# B&R Automation Studio project NAEUL004C00R13L518F00 (part 15)

#### Act_OptP0910WriteDO.st
```iecst
ACTION Act_OptP0910WriteDO:

	//TL Safety Relay
	IF tyP0910GenOut.tyGenOut.tyBtnSafetyRst.bRtCompl = TRUE THEN
		IF tyP0910GenOut.tyGenOut.tyBtnSafetyRst.bValue = TRUE THEN
			eRstErrAct	:= RstErrActSetSafetyRlyRst;

			IF p_eRstErrStat = RstErrActSetSafetyRlyRst AND p_eRstErrStatus = Done THEN
				eRstErrAct	:= RstErrActIdle;

				tyP0910GenOut.tyGenOut.tyBtnSafetyRst.bRtCompl	:= FALSE;
			END_IF
		ELSE
			eRstErrAct	:= RstErrActRstSafetyRlyRst;

			IF p_eRstErrStat = RstErrActRstSafetyRlyRst AND p_eRstErrStatus = Done THEN
				eRstErrAct	:= RstErrActIdle;

				tyP0910GenOut.tyGenOut.tyBtnSafetyRst.bRtCompl	:= FALSE;
			END_IF

		END_IF
	END_IF

	// TL Green
	IF tyP0910GenOut.tyGenOut.tyBtnTLGreen.bRtCompl = TRUE THEN
		IF tyP0910GenOut.tyGenOut.tyBtnTLGreen.bValue = TRUE THEN
			eTLBuzAct	:= TLBuzActSetGreen;

			IF p_eTLBuzStat = TLBuzActSetGreen AND p_eTLBuzStatus = Done THEN
				eTLBuzAct	:= TLBuzActIdle;

				tyP0910GenOut.tyGenOut.tyBtnTLGreen.bRtCompl	:= FALSE;
			END_IF
		ELSE
			eTLBuzAct	:= TLBuzActRstGreen;

			IF p_eTLBuzStat = TLBuzActRstGreen AND p_eTLBuzStatus = Done THEN
				eTLBuzAct	:= TLBuzActIdle;

				tyP0910GenOut.tyGenOut.tyBtnTLGreen.bRtCompl	:= FALSE;
			END_IF

		END_IF
	END_IF

	//TL Amber
	IF tyP0910GenOut.tyGenOut.tyBtnTLAmber.bRtCompl = TRUE THEN
		IF tyP0910GenOut.tyGenOut.tyBtnTLAmber.bValue = TRUE THEN
			IF p_tyNtParamCurr.eCustomerReq = Siemens THEN
				eTLBuzAct	:= TLBuzActSetWhite;
				IF p_eTLBuzStat = TLBuzActSetWhite AND p_eTLBuzStatus = Done THEN
					eTLBuzAct	:= TLBuzActIdle;
				END_IF
			ELSE
				eTLBuzAct	:= TLBuzActSetAmber;
				IF p_eTLBuzStat = TLBuzActSetAmber AND p_eTLBuzStatus = Done THEN
					eTLBuzAct	:= TLBuzActIdle;

					tyP0910GenOut.tyGenOut.tyBtnTLAmber.bRtCompl	:= FALSE;
				END_IF
			END_IF
		ELSE
			IF p_tyNtParamCurr.eCustomerReq = Siemens THEN
				eTLBuzAct	:= TLBuzActRstWhite;
				IF p_eTLBuzStat = TLBuzActRstWhite AND p_eTLBuzStatus = Done THEN
					eTLBuzAct	:= TLBuzActIdle;

					tyP0910GenOut.tyGenOut.tyBtnTLAmber.bRtCompl	:= FALSE;
				END_IF
			ELSE
				eTLBuzAct	:= TLBuzActRstAmber;
				IF p_eTLBuzStat = TLBuzActRstAmber AND p_eTLBuzStatus = Done THEN
					eTLBuzAct	:= TLBuzActIdle;

					tyP0910GenOut.tyGenOut.tyBtnTLAmber.bRtCompl	:= FALSE;
				END_IF
			END_IF
		END_IF
	END_IF

	//TL Red
	IF tyP0910GenOut.tyGenOut.tyBtnTLRed.bRtCompl = TRUE THEN
		IF tyP0910GenOut.tyGenOut.tyBtnTLRed.bValue = TRUE THEN
			eTLBuzAct	:= TLBuzActSetRed;

			IF p_eTLBuzStat = TLBuzActSetRed AND p_eTLBuzStatus = Done THEN
				eTLBuzAct	:= TLBuzActIdle;

				tyP0910GenOut.tyGenOut.tyBtnTLRed.bRtCompl	:= FALSE;
			END_IF
		ELSE
			eTLBuzAct	:= TLBuzActRstRed;

			IF p_eTLBuzStat = TLBuzActRstRed AND p_eTLBuzStatus = Done THEN
				eTLBuzAct	:= TLBuzActIdle;

				tyP0910GenOut.tyGenOut.tyBtnTLRed.bRtCompl	:= FALSE;
			END_IF

		END_IF
	END_IF

	//TL Buzzer
	IF tyP0910GenOut.tyGenOut.tyBtnBuzzer.bRtCompl = TRUE THEN
		IF tyP0910GenOut.tyGenOut.tyBtnBuzzer.bValue = TRUE THEN
			eTLBuzAct	:= TLBuzActSetBuz;

			IF p_eTLBuzStat = TLBuzActSetBuz AND p_eTLBuzStatus = Done THEN
				eTLBuzAct	:= TLBuzActIdle;

				tyP0910GenOut.tyGenOut.tyBtnBuzzer.bRtCompl	:= FALSE;
			END_IF
		ELSE
			eTLBuzAct	:= TLBuzActRstBuz;

			IF p_eTLBuzStat = TLBuzActRstBuz AND p_eTLBuzStatus = Done THEN
				eTLBuzAct	:= TLBuzActIdle;

				tyP0910GenOut.tyGenOut.tyBtnBuzzer.bRtCompl	:= FALSE;
			END_IF

		END_IF
	END_IF

	//Oven Info A
	IF tyP0910GenOut.tyOven.tyBtnOvenInfoA.bRtCompl = TRUE THEN
		IF tyP0910GenOut.tyOven.tyBtnOvenInfoA.bValue = TRUE THEN
			eOvenInfoAAct	:= OvenInfoActSetOvenAllow;

			IF p_eOvenInfoAStat = OvenInfoActSetOvenAllow AND p_eOvenInfoAStatus = Done THEN
				eOvenInfoAAct	:= OvenInfoActIdle;

				tyP0910GenOut.tyOven.tyBtnOvenInfoA.bRtCompl	:= FALSE;
			END_IF
		ELSE
			eOvenInfoAAct	:= OvenInfoActRstOvenAllow;

			IF p_eOvenInfoAStat = OvenInfoActRstOvenAllow AND p_eOvenInfoAStatus = Done THEN
				eOvenInfoAAct	:= OvenInfoActIdle;

				tyP0910GenOut.tyOven.tyBtnOvenInfoA.bRtCompl	:= FALSE;
			END_IF

		END_IF
	END_IF

	//Oven Info B
	IF tyP0910GenOut.tyOven.tyBtnOvenInfoB.bRtCompl = TRUE THEN
		IF tyP0910GenOut.tyOven.tyBtnOvenInfoB.bValue = TRUE THEN
			eOvenInfoBAct	:= OvenInfoActSetOvenAllow;

			IF p_eOvenInfoBStat = OvenInfoActSetOvenAllow AND p_eOvenInfoBStatus = Done THEN
				eOvenInfoBAct	:= OvenInfoActIdle;

				tyP0910GenOut.tyOven.tyBtnOvenInfoB.bRtCompl	:= FALSE;
			END_IF
		ELSE
			eOvenInfoBAct	:= OvenInfoActRstOvenAllow;

			IF p_eOvenInfoBStat = OvenInfoActRstOvenAllow AND p_eOvenInfoBStatus = Done THEN
				eOvenInfoBAct	:= OvenInfoActIdle;

				tyP0910GenOut.tyOven.tyBtnOvenInfoB.bRtCompl	:= FALSE;
			END_IF

		END_IF
	END_IF

	//Bypass Open Limit Sen
	IF tyP0910GenOut.tyMagAW.tyBtnMagAWOpenLimByp1.bRtCompl = TRUE THEN

		IF tyP0910GenOut.tyMagAW.tyBtnMagAWOpenLimByp1.bValue = TRUE THEN
			bMagAWOpenLimByp1 := TRUE;
			tyP0910GenOut.tyMagAW.tyBtnMagAWOpenLimByp1.bRtCompl := FALSE;
		ELSE
			bMagAWOpenLimByp1 := FALSE;
			tyP0910GenOut.tyMagAW.tyBtnMagAWOpenLimByp1.bRtCompl := FALSE;
		END_IF
	END_IF

	IF tyP0910GenOut.tyMagAW.tyBtnMagAWOpenLimByp2.bRtCompl = TRUE THEN

		IF tyP0910GenOut.tyMagAW.tyBtnMagAWOpenLimByp2.bValue = TRUE THEN
			bMagAWOpenLimByp2 := TRUE;
			tyP0910GenOut.tyMagAW.tyBtnMagAWOpenLimByp2.bRtCompl := FALSE;
		ELSE
			bMagAWOpenLimByp2 := FALSE;
			tyP0910GenOut.tyMagAW.tyBtnMagAWOpenLimByp2.bRtCompl := FALSE;
		END_IF
	END_IF

	IF tyP0910GenOut.tyMagAW.tyBtnMagAWOpenLimByp3.bRtCompl = TRUE THEN

		IF tyP0910GenOut.tyMagAW.tyBtnMagAWOpenLimByp3.bValue = TRUE THEN
			bMagAWOpenLimByp3 := TRUE;
			tyP0910GenOut.tyMagAW.tyBtnMagAWOpenLimByp3.bRtCompl := FALSE;
		ELSE
			bMagAWOpenLimByp3 := FALSE;
			tyP0910GenOut.tyMagAW.tyBtnMagAWOpenLimByp3.bRtCompl := FALSE;
		END_IF
	END_IF

	IF tyP0910GenOut.tyMagAW.tyBtnMagAWOpenLimByp4.bRtCompl = TRUE THEN

		IF tyP0910GenOut.tyMagAW.tyBtnMagAWOpenLimByp4.bValue = TRUE THEN
			bMagAWOpenLimByp4 := TRUE;
			tyP0910GenOut.tyMagAW.tyBtnMagAWOpenLimByp4.bRtCompl := FALSE;
		ELSE
			bMagAWOpenLimByp4 := FALSE;
			tyP0910GenOut.tyMagAW.tyBtnMagAWOpenLimByp4.bRtCompl := FALSE;
		END_IF
	END_IF

	//Select Small Mag Open Limit Sen
	IF tyP0910GenOut.tyMagAW.tyBtnSmallMagAWLimSen1.bRtCompl = TRUE THEN

		IF tyP0910GenOut.tyMagAW.tyBtnSmallMagAWLimSen1.bValue = TRUE THEN
			bSmallMagLimSen1 := TRUE;
			tyP0910GenOut.tyMagAW.tyBtnSmallMagAWLimSen1.bRtCompl := FALSE;
		ELSE
			bSmallMagLimSen1 := FALSE;
			tyP0910GenOut.tyMagAW.tyBtnSmallMagAWLimSen1.bRtCompl := FALSE;
		END_IF
	END_IF

	IF tyP0910GenOut.tyMagAW.tyBtnSmallMagAWLimSen2.bRtCompl = TRUE THEN

		IF tyP0910GenOut.tyMagAW.tyBtnSmallMagAWLimSen2.bValue = TRUE THEN
			bSmallMagLimSen2 := TRUE;
			tyP0910GenOut.tyMagAW.tyBtnSmallMagAWLimSen2.bRtCompl := FALSE;
		ELSE
			bSmallMagLimSen2 := FALSE;
			tyP0910GenOut.tyMagAW.tyBtnSmallMagAWLimSen2.bRtCompl := FALSE;
		END_IF
	END_IF

	IF tyP0910GenOut.tyMagAW.tyBtnSmallMagAWLimSen3.bRtCompl = TRUE THEN

		IF tyP0910GenOut.tyMagAW.tyBtnSmallMagAWLimSen3.bValue = TRUE THEN
			bSmallMagLimSen3 := TRUE;
			tyP0910GenOut.tyMagAW.tyBtnSmallMagAWLimSen3.bRtCompl := FALSE;
		ELSE
			bSmallMagLimSen3 := FALSE;
			tyP0910GenOut.tyMagAW.tyBtnSmallMagAWLimSen3.bRtCompl := FALSE;
		END_IF
	END_IF

	IF tyP0910GenOut.tyMagAW.tyBtnSmallMagAWLimSen4.bRtCompl = TRUE THEN

		IF tyP0910GenOut.tyMagAW.tyBtnSmallMagAWLimSen4.bValue = TRUE THEN
			bSmallMagLimSen4 := TRUE;
			tyP0910GenOut.tyMagAW.tyBtnSmallMagAWLimSen4.bRtCompl := FALSE;
		ELSE
			bSmallMagLimSen4 := FALSE;
			tyP0910GenOut.tyMagAW.tyBtnSmallMagAWLimSen4.bRtCompl := FALSE;
		END_IF
	END_IF

//	IF tyP0910GenOut.tyGenOutCurtainSen.tyBtnRstCurtainSen.bRtCompl = TRUE THEN
//
//		IF tyP0910GenOut.tyGenOutCurtainSen.tyBtnRstCurtainSen.bValue = TRUE THEN
//			bSafetyCurtainReset := TRUE;
//			tyP0910GenOut.tyGenOutCurtainSen.tyBtnRstCurtainSen.bRtCompl := FALSE;
//		ELSE
//			bSafetyCurtainReset := FALSE;
//			tyP0910GenOut.tyGenOutCurtainSen.tyBtnRstCurtainSen.bRtCompl := FALSE;
//		END_IF
//	END_IF

	bBypCurtainPBLED	:= tyP0910GenOut.tyGenOutCurtainSen.tyBtnBypCurtainSenPBLED.bValue;
	bBypCurtainSen		:= tyP0910GenOut.tyGenOutCurtainSen.tyBtnBypCurtainSen.bValue;

END_ACTION
```

#### Act_OptP0910RstMnl.st
```iecst
ACTION Act_OptP0910RstMnl:

	IF EDGEPOS((bUIManualMod = FALSE) OR (p_eRstErrStatus = Error)) THEN
		eRstErrAct	:= RstErrActIdle;

		tyP0910GenOut.tyGenOut.tyBtnSafetyRst.bValue	:= FALSE;
	END_IF

	IF EDGEPOS((bUIManualMod = FALSE) OR (p_eTLBuzStatus = Error)) THEN
		eTLBuzAct	:= TLBuzActIdle;

		tyP0910GenOut.tyGenOut.tyBtnTLGreen.bValue		:= FALSE;
		tyP0910GenOut.tyGenOut.tyBtnTLAmber.bValue		:= FALSE;
		tyP0910GenOut.tyGenOut.tyBtnTLRed.bValue		:= FALSE;
		tyP0910GenOut.tyGenOut.tyBtnBuzzer.bValue		:= FALSE;
	END_IF

	IF EDGEPOS((bUIManualMod = FALSE) OR (p_eOvenInfoAStatus = Error)) THEN
		eOvenInfoAAct	:= OvenInfoActIdle;

		tyP0910GenOut.tyOven.tyBtnOvenInfoA.bValue	:= FALSE;
	END_IF

	IF EDGEPOS((bUIManualMod = FALSE) OR (p_eOvenInfoAStatus = Error)) THEN
		eOvenInfoBAct	:= OvenInfoActIdle;

		tyP0910GenOut.tyOven.tyBtnOvenInfoB.bValue	:= FALSE;
	END_IF

	IF EDGEPOS(bUIManualMod = FALSE)
		THEN
		tyP0910GenOut.tyMagAW.tyBtnMagAWOpenLimByp1.bValue 				:= FALSE;
		tyP0910GenOut.tyMagAW.tyBtnMagAWOpenLimByp2.bValue				:= FALSE;
		tyP0910GenOut.tyMagAW.tyBtnMagAWOpenLimByp3.bValue 				:= FALSE;
		tyP0910GenOut.tyMagAW.tyBtnMagAWOpenLimByp4.bValue 				:= FALSE;
		tyP0910GenOut.tyMagAW.tyBtnSmallMagAWLimSen1.bValue 			:= FALSE;
		tyP0910GenOut.tyMagAW.tyBtnSmallMagAWLimSen2.bValue 			:= FALSE;
		tyP0910GenOut.tyMagAW.tyBtnSmallMagAWLimSen3.bValue 			:= FALSE;
		tyP0910GenOut.tyMagAW.tyBtnSmallMagAWLimSen4.bValue 			:= FALSE;

		//Bypass Curtain Sensor and LED Display
		tyP0910GenOut.tyGenOutCurtainSen.tyBtnBypCurtainSenPBLED.bValue	:= FALSE;
		tyP0910GenOut.tyGenOutCurtainSen.tyBtnBypCurtainSen.bValue		:= FALSE;

		//Variable Data
		bBypCurtainSen		:= FALSE;
		bBypCurtainPBLED	:= FALSE;

		bMagAWOpenLimByp1 	:= FALSE;
		bMagAWOpenLimByp2 	:= FALSE;
		bMagAWOpenLimByp3	:= FALSE;
		bMagAWOpenLimByp4 	:= FALSE;
		bSmallMagLimSen1	:= FALSE;
		bSmallMagLimSen2	:= FALSE;
		bSmallMagLimSen3	:= FALSE;
		bSmallMagLimSen4	:= FALSE;

	END_IF

//	tyP0910GenOut.tyGenOutCurtainSen.tyBtnRstCurtainSen.bRtCompl	:= FALSE;
//	tyP0910GenOut.tyGenOutCurtainSen.tyBtnRstCurtainSen.bValue   	:= FALSE;
//	bSafetyCurtainReset	:= FALSE;

END_ACTION
```

#### Act_EntP0920Disp.st
```iecst
ACTION Act_EntP0920Disp:

	//Access Address
	p_tyC0002FullMask ACCESS ADR(tyP0920MtrNPneuCtrl.tyFullMaskHide);

	p_tyC0005Main ACCESS ADR(tyCommon.tyMain);

	p_tyC0007Notif ACCESS ADR(tyCommon.tyNotif);

	p_tyC0008MsgBox ACCESS ADR(tyP0920MtrNPneuCtrl.tyMsgBoxHide);

	p_tyC0009Info ACCESS ADR(tyCommon.tyInfo);

	p_tyP0920MtrNPneuCtrl ACCESS ADR(tyP0920MtrNPneuCtrl.tyMtrNPneuCtrl);

	p_tyP0920MtrNPneuCtrlPneu ACCESS ADR(tyP0920MtrNPneuCtrl.tyMtrNPneuCtrlPneu);

	//Display
	//Auto Width
	tyP0920MtrNPneuCtrl.tyMtrNPneuCtrl.tyBtnAW.uiMaskRtStat.0	:= NOT(p_tyNtParamCurr.bAWPrep AND p_tyMcParamCurr.bAWDis);
	tyP0920MtrNPneuCtrl.tyMtrNPneuCtrl.tyBtnAWPushPul.uiMaskRtStat.0	:= NOT(p_tyNtParamCurr.bAWPusherPrep AND p_tyMcParamCurr.bAWPusherDis);
	//Magazine Auto Width
	tyP0920MtrNPneuCtrl.tyMtrNPneuCtrl.tyBtnMagAW.uiMaskRtStat.0	:= NOT(p_tyNtParamCurr.bProjMagAWPrep AND p_tyMcParamCurr.bMagAWDis);

END_ACTION
```

#### Act_OptP0920FullMask.st
```iecst
ACTION Act_OptP0920FullMask:

	IF eCurrPage = UIP0920MtrNPneuCtrl THEN

		IF p_tyDI.bEStopSig = FALSE THEN
			p_tyC0002FullMask ACCESS ADR(tyP0920MtrNPneuCtrl.tyFullMaskEStop);

		ELSIF p_tyDI.bCoverSWSig = FALSE THEN
			p_tyC0002FullMask ACCESS ADR(tyP0920MtrNPneuCtrl.tyFullMaskCWSig);

		ELSIF p_tyDI.bSafetyRlySig = FALSE THEN
			p_tyC0002FullMask ACCESS ADR(tyP0920MtrNPneuCtrl.tyFullMaskSafetyRly);

		ELSE
			p_tyC0002FullMask ACCESS ADR(tyP0920MtrNPneuCtrl.tyFullMaskHide);

		END_IF

	END_IF

END_ACTION
```

#### Act_OptP0920ChgPage.st
```iecst
ACTION Act_OptP0920ChgPage:

	IF tyP0920MtrNPneuCtrl.tyMtrNPneuCtrlPneu.tyBtnShutter.bRtCompl THEN
		tyP0920MtrNPneuCtrl.tyMtrNPneuCtrlPneu.tyBtnShutter.bRtCompl	:= FALSE;
		tyP0920MtrNPneuCtrl.tyMtrNPneuCtrlPneu.tyBtnShutter.bValue		:= FALSE;
		eChgPage														:= UIP0921Shutter;

	ELSIF tyP0920MtrNPneuCtrl.tyMtrNPneuCtrlPneu.tyBtnStopper.bRtCompl THEN
		tyP0920MtrNPneuCtrl.tyMtrNPneuCtrlPneu.tyBtnStopper.bRtCompl	:= FALSE;
		tyP0920MtrNPneuCtrl.tyMtrNPneuCtrlPneu.tyBtnStopper.bValue		:= FALSE;
		eChgPage														:= UIP0922Stopper;

	ELSIF tyP0920MtrNPneuCtrl.tyMtrNPneuCtrl.tyBtnLifterConv.bRtCompl AND p_tyNtParamCurr.bProjMagConvLane1Prep THEN
		tyP0920MtrNPneuCtrl.tyMtrNPneuCtrl.tyBtnLifterConv.bRtCompl		:= FALSE;
		tyP0920MtrNPneuCtrl.tyMtrNPneuCtrl.tyBtnLifterConv.bValue		:= FALSE;
		eChgPage														:= UIP0926LifterConv;

	ELSIF tyP0920MtrNPneuCtrl.tyMtrNPneuCtrl.tyBtnLifterConv2.bRtCompl AND p_tyNtParamCurr.bProjMagConvLane2Prep THEN
		tyP0920MtrNPneuCtrl.tyMtrNPneuCtrl.tyBtnLifterConv2.bRtCompl		:= FALSE;
		tyP0920MtrNPneuCtrl.tyMtrNPneuCtrl.tyBtnLifterConv2.bValue			:= FALSE;
		eChgPage														:= UIP0927LifterConv2;

	ELSIF tyP0920MtrNPneuCtrl.tyMtrNPneuCtrl.tyBtnMag1Conv.bRtCompl AND p_tyNtParamCurr.bProjMagConvLane1Prep THEN
		tyP0920MtrNPneuCtrl.tyMtrNPneuCtrl.tyBtnMag1Conv.bRtCompl		:= FALSE;
		tyP0920MtrNPneuCtrl.tyMtrNPneuCtrl.tyBtnMag1Conv.bValue			:= FALSE;
		eChgPage														:= UIP0928MagConv;

	ELSIF tyP0920MtrNPneuCtrl.tyMtrNPneuCtrl.tyBtnMag1Conv.bRtCompl AND bDispMagConv1 AND NOT(p_tyNtParamCurr.bProjMagConvLane1Prep) THEN
		tyP0920MtrNPneuCtrl.tyMtrNPneuCtrl.tyBtnMag1Conv.bRtCompl		:= FALSE;
		tyP0920MtrNPneuCtrl.tyMtrNPneuCtrl.tyBtnMag1Conv.bValue			:= FALSE;
		eChgPage														:= UIP0930MagConv1;

	ELSIF tyP0920MtrNPneuCtrl.tyMtrNPneuCtrl.tyBtnMag1Conv.bRtCompl AND bDispMagConv2 THEN
		tyP0920MtrNPneuCtrl.tyMtrNPneuCtrl.tyBtnMag1Conv.bRtCompl		:= FALSE;
		tyP0920MtrNPneuCtrl.tyMtrNPneuCtrl.tyBtnMag1Conv.bValue			:= FALSE;
		eChgPage														:= UIP0931MagConv2;

	ELSIF tyP0920MtrNPneuCtrl.tyMtrNPneuCtrl.tyBtnMag1Conv.bRtCompl AND bDispMagConv3 THEN
		tyP0920MtrNPneuCtrl.tyMtrNPneuCtrl.tyBtnMag1Conv.bRtCompl		:= FALSE;
		tyP0920MtrNPneuCtrl.tyMtrNPneuCtrl.tyBtnMag1Conv.bValue			:= FALSE;
		eChgPage														:= UIP0932MagConv3;

	ELSIF tyP0920MtrNPneuCtrl.tyMtrNPneuCtrl.tyBtnPusherConv.bRtCompl = TRUE THEN
		tyP0920MtrNPneuCtrl.tyMtrNPneuCtrl.tyBtnPusherConv.bRtCompl		:= FALSE;
		tyP0920MtrNPneuCtrl.tyMtrNPneuCtrl.tyBtnPusherConv.bValue		:= FALSE;
		eChgPage														:= UIP0933PusherConv;

	ELSIF tyP0920MtrNPneuCtrl.tyMtrNPneuCtrl.tyBtnAW.bRtCompl = TRUE THEN
		tyP0920MtrNPneuCtrl.tyMtrNPneuCtrl.tyBtnAW.bRtCompl				:= FALSE;
		tyP0920MtrNPneuCtrl.tyMtrNPneuCtrl.tyBtnAW.bValue				:= FALSE;
		eChgPage														:= UIP0934AW;

	ELSIF tyP0920MtrNPneuCtrl.tyMtrNPneuCtrl.tyBtnLifter.bRtCompl = TRUE THEN
		tyP0920MtrNPneuCtrl.tyMtrNPneuCtrl.tyBtnLifter.bRtCompl			:= FALSE;
		tyP0920MtrNPneuCtrl.tyMtrNPneuCtrl.tyBtnLifter.bValue			:= FALSE;
		eChgPage														:= UIP0935Lifter;

	ELSIF tyP0920MtrNPneuCtrl.tyMtrNPneuCtrl.tyBtnTrav.bRtCompl = TRUE THEN
		tyP0920MtrNPneuCtrl.tyMtrNPneuCtrl.tyBtnTrav.bRtCompl			:= FALSE;
		tyP0920MtrNPneuCtrl.tyMtrNPneuCtrl.tyBtnTrav.bValue				:= FALSE;
		eChgPage														:= UIP0936Trav;

	ELSIF tyP0920MtrNPneuCtrl.tyMtrNPneuCtrl.tyBtnMagAW.bRtCompl = TRUE THEN
		tyP0920MtrNPneuCtrl.tyMtrNPneuCtrl.tyBtnMagAW.bRtCompl			:= FALSE;
		tyP0920MtrNPneuCtrl.tyMtrNPneuCtrl.tyBtnMagAW.bValue			:= FALSE;
		eChgPage														:= UIP0938MagAW;

	ELSIF tyP0920MtrNPneuCtrl.tyMtrNPneuCtrl.tyBtnLifter2.bRtCompl THEN
		tyP0920MtrNPneuCtrl.tyMtrNPneuCtrl.tyBtnLifter2.bRtCompl	:= FALSE;
		tyP0920MtrNPneuCtrl.tyMtrNPneuCtrl.tyBtnLifter2.bValue		:= FALSE;
		eChgPage													:= UIP0939Lifter2;

	ELSIF tyP0920MtrNPneuCtrl.tyMtrNPneuCtrl.tyBtnAWPushPul.bRtCompl = TRUE THEN
		tyP0920MtrNPneuCtrl.tyMtrNPneuCtrl.tyBtnAWPushPul.bRtCompl		:= FALSE;
		tyP0920MtrNPneuCtrl.tyMtrNPneuCtrl.tyBtnAWPushPul.bValue		:= FALSE;
		eChgPage														:= UIP0937AWPushOrPuller;

	ELSIF tyP0920MtrNPneuCtrl.tyMtrNPneuCtrlPneu.tyBtnSafetyBar.bRtCompl THEN
		tyP0920MtrNPneuCtrl.tyMtrNPneuCtrlPneu.tyBtnSafetyBar.bRtCompl	:= FALSE;
		tyP0920MtrNPneuCtrl.tyMtrNPneuCtrlPneu.tyBtnSafetyBar.bValue	:= FALSE;
		eChgPage														:= UIP0923SafetyBar;
	END_IF

END_ACTION
```

#### Act_EntP0921Disp.st
```iecst
ACTION Act_EntP0921Disp:

	//Access Address
	p_tyC0003DualMask ACCESS ADR(tyP0921InletNOutletShutter.tyDualMaskHide);

	//Add_2022.12.12
	IF NOT p_tyNtParamCurr.bProjOutletShut2Prep OR NOT p_tyNtParamCurr.bProjOutletShut3Prep THEN
		p_tyC0004Navi ACCESS ADR (tyP0921InletNOutletShutter.tyNaviBack);
	ELSE
		p_tyC0004Navi ACCESS ADR (tyP0921InletNOutletShutter.tyNaviLyr1);
	END_IF

	//	p_tyC0004Navi ACCESS ADR(tyP0921InletNOutletShutter.tyNaviBack);
	//	p_tyC0004Navi ACCESS ADR(tyP0921InletNOutletShutter.tyNaviLyr1);

	p_tyC0005Main ACCESS ADR(tyCommon.tyMain);

	p_tyC0007Notif ACCESS ADR(tyCommon.tyNotif);

	p_tyC0008MsgBox ACCESS ADR(tyP0921InletNOutletShutter.tyMsgBoxHide);

	p_tyC0009Info ACCESS ADR(tyCommon.tyInfo);

	p_tyP0921InletShutterCom ACCESS ADR(tyP0921InletNOutletShutter.tyInletShutterCom);
	p_tyP0921InletShutterDC ACCESS ADR(tyP0921InletNOutletShutter.tyInletShutterDC);
	p_tyP0921InletShutterFB ACCESS ADR(tyP0921InletNOutletShutter.tyInletShutterFB);
	p_tyP0921InletShutterDis ACCESS ADR(tyP0921InletNOutletShutter.tyInletShutterDis);

	p_tyP0921OutletShutterCom ACCESS ADR(tyP0921InletNOutletShutter.tyOutletShutterCom);
	p_tyP0921OutletShutterDC ACCESS ADR(tyP0921InletNOutletShutter.tyOutletShutterDC);
	p_tyP0921OutletShutterFB ACCESS ADR(tyP0921InletNOutletShutter.tyOutletShutterFB);

	//Display
//	tyP0921InletNOutletShutter.tyInletShutterDis.tyLyr.uiRtStat.0	:= NOT(p_tyNtParamCurr.bProjInletShutPrep AND p_tyMcParamCurr.bInShutterDis);

END_ACTION
```

#### Act_OptP0921Navi.st
```iecst
ACTION Act_OptP0921Navi:

	IF tyP0921InletNOutletShutter.tyNaviLyr1.tyBtnBack.bRtCompl = TRUE OR tyP0921InletNOutletShutter.tyNaviLyr2.tyBtnBack.bRtCompl = TRUE OR
		 tyP0921InletNOutletShutter.tyNaviBack.tyBtnBack.bRtCompl = TRUE THEN

		eChgPage		:= UIP0920MtrNPneuCtrl;

		tyP0921InletNOutletShutter.tyNaviLyr1.tyBtnBack.bRtCompl := FALSE;
		tyP0921InletNOutletShutter.tyNaviLyr1.tyBtnBack.bValue	 := FALSE;

		tyP0921InletNOutletShutter.tyNaviLyr2.tyBtnBack.bRtCompl := FALSE;
		tyP0921InletNOutletShutter.tyNaviLyr2.tyBtnBack.bValue	 := FALSE;

		tyP0921InletNOutletShutter.tyNaviBack.tyBtnBack.bRtCompl := FALSE;
		tyP0921InletNOutletShutter.tyNaviBack.tyBtnBack.bValue	 := FALSE;

	ELSIF tyP0921InletNOutletShutter.tyNaviLyr1.tyBtnRgt.bRtCompl THEN

		p_tyC0004Navi ACCESS ADR (tyP0921InletNOutletShutter.tyNaviLyr2);

		p_tyP0921InletShutterCom ACCESS ADR(tyP0921InletNOutletShutter.tyOutletShutterCom2);
		p_tyP0921InletShutterDC ACCESS ADR(tyP0921InletNOutletShutter.tyOutletShutterDC2);
		p_tyP0921InletShutterFB ACCESS ADR(tyP0921InletNOutletShutter.tyOutletShutterFB2);
		p_tyP0921InletShutterDis ACCESS ADR(tyP0921InletNOutletShutter.tyOutletShutterDis2);

		p_tyP0921OutletShutterCom ACCESS ADR(tyP0921InletNOutletShutter.tyOutletShutterCom3);
		p_tyP0921OutletShutterDC ACCESS ADR(tyP0921InletNOutletShutter.tyOutletShutterDC3);
		p_tyP0921OutletShutterFB ACCESS ADR(tyP0921InletNOutletShutter.tyOutletShutterFB3);

		tyP0921InletNOutletShutter.tyNaviLyr1.tyBtnRgt.bRtCompl := FALSE;

	ELSIF tyP0921InletNOutletShutter.tyNaviLyr1.tyBtnLeft.bRtCompl THEN

		p_tyC0004Navi ACCESS ADR (tyP0921InletNOutletShutter.tyNaviLyr2);

		p_tyP0921InletShutterCom ACCESS ADR(tyP0921InletNOutletShutter.tyOutletShutterCom2);
		p_tyP0921InletShutterDC ACCESS ADR(tyP0921InletNOutletShutter.tyOutletShutterDC2);
		p_tyP0921InletShutterFB ACCESS ADR(tyP0921InletNOutletShutter.tyOutletShutterFB2);
		p_tyP0921InletShutterDis ACCESS ADR(tyP0921InletNOutletShutter.tyOutletShutterDis2);

		p_tyP0921OutletShutterCom ACCESS ADR(tyP0921InletNOutletShutter.tyOutletShutterCom3);
		p_tyP0921OutletShutterDC ACCESS ADR(tyP0921InletNOutletShutter.tyOutletShutterDC3);
		p_tyP0921OutletShutterFB ACCESS ADR(tyP0921InletNOutletShutter.tyOutletShutterFB3);

		tyP0921InletNOutletShutter.tyNaviLyr1.tyBtnLeft.bRtCompl := FALSE;

	ELSIF tyP0921InletNOutletShutter.tyNaviLyr2.tyBtnRgt.bRtCompl THEN

		p_tyC0004Navi ACCESS ADR (tyP0921InletNOutletShutter.tyNaviLyr1);

		p_tyP0921InletShutterCom ACCESS ADR(tyP0921InletNOutletShutter.tyInletShutterCom);
		p_tyP0921InletShutterDC ACCESS ADR(tyP0921InletNOutletShutter.tyInletShutterDC);
		p_tyP0921InletShutterFB ACCESS ADR(tyP0921InletNOutletShutter.tyInletShutterFB);
		p_tyP0921InletShutterDis ACCESS ADR(tyP0921InletNOutletShutter.tyInletShutterDis);

		p_tyP0921OutletShutterCom ACCESS ADR(tyP0921InletNOutletShutter.tyOutletShutterCom);
		p_tyP0921OutletShutterDC ACCESS ADR(tyP0921InletNOutletShutter.tyOutletShutterDC);
		p_tyP0921OutletShutterFB ACCESS ADR(tyP0921InletNOutletShutter.tyOutletShutterFB);

		tyP0921InletNOutletShutter.tyNaviLyr2.tyBtnRgt.bRtCompl := FALSE;

	ELSIF tyP0921InletNOutletShutter.tyNaviLyr2.tyBtnLeft.bRtCompl THEN

		p_tyC0004Navi ACCESS ADR (tyP0921InletNOutletShutter.tyNaviLyr1);

		p_tyP0921InletShutterCom ACCESS ADR(tyP0921InletNOutletShutter.tyInletShutterCom);
		p_tyP0921InletShutterDC ACCESS ADR(tyP0921InletNOutletShutter.tyInletShutterDC);
		p_tyP0921InletShutterFB ACCESS ADR(tyP0921InletNOutletShutter.tyInletShutterFB);
		p_tyP0921InletShutterDis ACCESS ADR(tyP0921InletNOutletShutter.tyInletShutterDis);

		p_tyP0921OutletShutterCom ACCESS ADR(tyP0921InletNOutletShutter.tyOutletShutterCom);
		p_tyP0921OutletShutterDC ACCESS ADR(tyP0921InletNOutletShutter.tyOutletShutterDC);
		p_tyP0921OutletShutterFB ACCESS ADR(tyP0921InletNOutletShutter.tyOutletShutterFB);

		tyP0921InletNOutletShutter.tyNaviLyr2.tyBtnLeft.bRtCompl := FALSE;

	END_IF

END_ACTION
```

#### Act_OptP0921DualMask.st
```iecst
ACTION Act_OptP0921DualMask:

	IF eCurrPage = UIP0921Shutter THEN

		IF p_tyDI.bEStopSig = FALSE THEN
			p_tyC0003DualMask ACCESS ADR(tyP0921InletNOutletShutter.tyDualMaskEStop);

			tyP0921InletNOutletShutter.tyDualMaskEStop.tyBtnLeftMask.uiMaskRtStat.0	:= NOT p_tyNtParamCurr.bProjInletShutPrep;
			tyP0921InletNOutletShutter.tyDualMaskEStop.tyBtnRgtMask.uiMaskRtStat.0	:= NOT p_tyNtParamCurr.bProjOutletShutPrep;

		ELSIF p_tyDI.bCoverSWSig = FALSE THEN
			p_tyC0003DualMask ACCESS ADR(tyP0921InletNOutletShutter.tyDualMaskCWSig);

			tyP0921InletNOutletShutter.tyDualMaskCWSig.tyBtnLeftMask.uiMaskRtStat.0	:= NOT p_tyNtParamCurr.bProjInletShutPrep;
			tyP0921InletNOutletShutter.tyDualMaskCWSig.tyBtnRgtMask.uiMaskRtStat.0	:= NOT p_tyNtParamCurr.bProjOutletShutPrep;

		ELSIF p_tyDI.bSafetyRlySig = FALSE THEN
			p_tyC0003DualMask ACCESS ADR(tyP0921InletNOutletShutter.tyDualMaskSafetyRly);

			tyP0921InletNOutletShutter.tyDualMaskSafetyRly.tyBtnLeftMask.uiMaskRtStat.0	:= NOT p_tyNtParamCurr.bProjInletShutPrep;
			tyP0921InletNOutletShutter.tyDualMaskSafetyRly.tyBtnRgtMask.uiMaskRtStat.0	:= NOT p_tyNtParamCurr.bProjOutletShutPrep;

		ELSIF p_eLifterBtmStatus = Busy AND p_bLifterBtmPwrOn THEN
			p_tyC0003DualMask ACCESS ADR(tyP0921InletNOutletShutter.tyDualMaskLifMovInterrupt);

			tyP0921InletNOutletShutter.tyDualMaskLifMovInterrupt.tyBtnLeftMask.uiMaskRtStat.0	:= NOT p_tyNtParamCurr.bProjInletShutPrep;
			tyP0921InletNOutletShutter.tyDualMaskLifMovInterrupt.tyBtnRgtMask.uiMaskRtStat.0	:= NOT p_tyNtParamCurr.bProjOutletShutPrep;

		ELSIF p_eTravStatus = Busy AND p_bTravPwrOn THEN
			p_tyC0003DualMask ACCESS ADR(tyP0921InletNOutletShutter.tyDualMaskTravMovInterrupt);

			tyP0921InletNOutletShutter.tyDualMaskTravMovInterrupt.tyBtnLeftMask.uiMaskRtStat.0	:= NOT p_tyNtParamCurr.bProjInletShutPrep;
			tyP0921InletNOutletShutter.tyDualMaskTravMovInterrupt.tyBtnRgtMask.uiMaskRtStat.0	:= NOT p_tyNtParamCurr.bProjOutletShutPrep;

		ELSIF p_eAWOpenStatus = Busy AND p_bAWOpenPwrOn THEN
			p_tyC0003DualMask ACCESS ADR(tyP0921InletNOutletShutter.tyDualMaskAWMovInterrupt);

			tyP0921InletNOutletShutter.tyDualMaskAWMovInterrupt.tyBtnLeftMask.uiMaskRtStat.0	:= NOT p_tyNtParamCurr.bProjInletShutPrep;
			tyP0921InletNOutletShutter.tyDualMaskAWMovInterrupt.tyBtnRgtMask.uiMaskRtStat.0		:= NOT p_tyNtParamCurr.bProjOutletShutPrep;

		ELSIF p_tyDI.bPusherRetRS = FALSE THEN
			IF p_tyC0004Navi.tyBitmapPageDisp.usiValueIdx = 1 THEN
				p_tyC0003DualMask ACCESS ADR(tyP0921InletNOutletShutter.tyDualMaskPshrInterruptInOutlet);
			ELSIF p_tyC0004Navi.tyBitmapPageDisp.usiValueIdx = 2 THEN
				p_tyC0003DualMask ACCESS ADR(tyP0921InletNOutletShutter.tyDualMaskPshrInterruptOutlet);
			END_IF
		ELSE
			p_tyC0003DualMask ACCESS ADR(tyP0921InletNOutletShutter.tyDualMaskHide);
		END_IF

	END_IF

END_ACTION
```

#### Act_OptP0921InletShutterChgLyr.st
```iecst
ACTION Act_OptP0921InletShutterChgLyr:

	IF tyP0921InletNOutletShutter.tyInletShutterCom.tyBtnSwitch.bRtCompl THEN
		tyP0921InletNOutletShutter.tyInletShutterCom.tyBtnSwitch.bRtCompl := FALSE;

		IF tyP0921InletNOutletShutter.tyInletShutterCom.tyBtnSwitch.bValue = TRUE THEN
			fUIInRtStatOff(ADR(tyP0921InletNOutletShutter.tyInletShutterDC.tyLyr.uiRtStat));
			fUIInRtStatHide(ADR(tyP0921InletNOutletShutter.tyInletShutterFB.tyLyr.uiRtStat));
		ELSE
			fUIInRtStatHide(ADR(tyP0921InletNOutletShutter.tyInletShutterDC.tyLyr.uiRtStat));
			fUIInRtStatOff(ADR(tyP0921InletNOutletShutter.tyInletShutterFB.tyLyr.uiRtStat));
		END_IF

	END_IF

END_ACTION
```

#### Act_OptP0921InletShutterSen.st
```iecst
ACTION Act_OptP0921InletShutterSen:

	tyP0921InletNOutletShutter.tyInletShutterCom.tyBtnOpenRS.bValue		:= p_tyDI.bInShutterOpenRS;
	tyP0921InletNOutletShutter.tyInletShutterCom.tyBtnCloseRS.bValue	:= p_tyDI.bInShutterCloseRS;

	//Machine Bitmap
	IF p_tyDI.bInShutterOpenRS = TRUE THEN
		tyP0921InletNOutletShutter.tyInletShutterCom.tyBitmapMc.uiValueIdx	:= 1;
	ELSE
		tyP0921InletNOutletShutter.tyInletShutterCom.tyBitmapMc.uiValueIdx	:= 0;
	END_IF

	IF p_tyNtParamCurr.eProjMag = ULMagTriple THEN
		IF p_tyNtParamCurr.bProjLifterMagPlatform AND p_tyNtParamCurr.bUIConvDirRL THEN
			IF 	tyP0921InletNOutletShutter.tyInletShutterCom.tyBitmapMc.uiValueIdx < 100 THEN
				tyP0921InletNOutletShutter.tyInletShutterCom.tyBitmapMc.uiValueIdx	:= tyP0921InletNOutletShutter.tyInletShutterCom.tyBitmapMc.uiValueIdx + 800;
			END_IF
		ELSIF p_tyNtParamCurr.bProjLifterMagPlatform THEN
			IF 	tyP0921InletNOutletShutter.tyInletShutterCom.tyBitmapMc.uiValueIdx < 100 THEN
				tyP0921InletNOutletShutter.tyInletShutterCom.tyBitmapMc.uiValueIdx	:= tyP0921InletNOutletShutter.tyInletShutterCom.tyBitmapMc.uiValueIdx + 500;
			END_IF
		ELSIF p_tyNtParamCurr.bProjMagAWPrep = FALSE AND p_tyNtParamCurr.bProjMagSafetyBarPrep = FALSE THEN
			IF 	tyP0921InletNOutletShutter.tyInletShutterCom.tyBitmapMc.uiValueIdx < 100 THEN
				tyP0921InletNOutletShutter.tyInletShutterCom.tyBitmapMc.uiValueIdx	:= tyP0921InletNOutletShutter.tyInletShutterCom.tyBitmapMc.uiValueIdx + 100;
			END_IF

		ELSIF p_tyNtParamCurr.eProjMag = ULMagTriple AND p_tyNtParamCurr.bProjMagAWPrep THEN
				IF 	tyP0921InletNOutletShutter.tyInletShutterCom.tyBitmapMc.uiValueIdx < 134 THEN
					tyP0921InletNOutletShutter.tyInletShutterCom.tyBitmapMc.uiValueIdx	:= tyP0921InletNOutletShutter.tyInletShutterCom.tyBitmapMc.uiValueIdx + 134;
				END_IF

		ELSIF p_tyNtParamCurr.bProjMagAWPrep = FALSE AND p_tyNtParamCurr.bProjMagSafetyBarPrep = TRUE THEN
			IF 	tyP0921InletNOutletShutter.tyInletShutterCom.tyBitmapMc.uiValueIdx < 402 THEN
				tyP0921InletNOutletShutter.tyInletShutterCom.tyBitmapMc.uiValueIdx	:= tyP0921InletNOutletShutter.tyInletShutterCom.tyBitmapMc.uiValueIdx + 402;
			END_IF
		END_IF
	ELSIF p_tyNtParamCurr.eProjMag = ULMagDual THEN
		IF p_tyNtParamCurr.bProjLifterMagPlatform AND p_tyNtParamCurr.bUIConvDirRL THEN
			IF 	tyP0921InletNOutletShutter.tyInletShutterCom.tyBitmapMc.uiValueIdx < 100 THEN
				tyP0921InletNOutletShutter.tyInletShutterCom.tyBitmapMc.uiValueIdx	:= tyP0921InletNOutletShutter.tyInletShutterCom.tyBitmapMc.uiValueIdx + 700;
			END_IF
		ELSIF p_tyNtParamCurr.bProjLifterMagPlatform AND p_tyNtParamCurr.bUIConvDirRL = FALSE AND p_tyNtParamCurr.bProjMagConvLane1Prep THEN
			IF 	tyP0921InletNOutletShutter.tyInletShutterCom.tyBitmapMc.uiValueIdx < 100 THEN
				tyP0921InletNOutletShutter.tyInletShutterCom.tyBitmapMc.uiValueIdx	:= tyP0921InletNOutletShutter.tyInletShutterCom.tyBitmapMc.uiValueIdx + 900;
			END_IF
		ELSIF p_tyNtParamCurr.bProjLifterMagPlatform THEN
			IF 	tyP0921InletNOutletShutter.tyInletShutterCom.tyBitmapMc.uiValueIdx < 100 THEN
				tyP0921InletNOutletShutter.tyInletShutterCom.tyBitmapMc.uiValueIdx	:= tyP0921InletNOutletShutter.tyInletShutterCom.tyBitmapMc.uiValueIdx + 600;
			END_IF
		ELSIF p_tyNtParamCurr.bProjMagAWPrep = FALSE THEN
			tyP0921InletNOutletShutter.tyInletShutterCom.tyBitmapMc.uiValueIdx	:= tyP0921InletNOutletShutter.tyInletShutterCom.tyBitmapMc.uiValueIdx + 200;
		ELSIF p_tyNtParamCurr.bProjMagAWPrep THEN
			tyP0921InletNOutletShutter.tyInletShutterCom.tyBitmapMc.uiValueIdx	:= tyP0921InletNOutletShutter.tyInletShutterCom.tyBitmapMc.uiValueIdx + 334;
		END_IF
	END_IF
END_ACTION
```

#### Act_OptP0921InletShutterFB.st
```iecst
ACTION Act_OptP0921InletShutterFB:

	IF tyP0921InletNOutletShutter.tyInletShutterCom.tyBtnSwitch.bValue = FALSE THEN

		IF tyP0921InletNOutletShutter.tyInletShutterFB.tyBtnOpen.bRtCompl = TRUE THEN
			tyP0921InletNOutletShutter.tyInletShutterFB.tyBtnOpen.bRtCompl	:= FALSE;

			tyP0921InletNOutletShutter.tyInletShutterFB.tyBtnOpen.bValue	:= TRUE;
			tyP0921InletNOutletShutter.tyInletShutterFB.tyBtnClose.bValue	:= FALSE;

		ELSIF tyP0921InletNOutletShutter.tyInletShutterFB.tyBtnClose.bRtCompl = TRUE THEN
			tyP0921InletNOutletShutter.tyInletShutterFB.tyBtnClose.bRtCompl	:= FALSE;

			tyP0921InletNOutletShutter.tyInletShutterFB.tyBtnClose.bValue	:= TRUE;
			tyP0921InletNOutletShutter.tyInletShutterFB.tyBtnOpen.bValue	:= FALSE;
		END_IF

		IF tyP0921InletNOutletShutter.tyInletShutterFB.tyBtnOpen.bValue = TRUE THEN
			eInShutterAct	:= PneuActRet;

			IF p_eInShutterStat = PneuActRet AND p_eInShutterStatus = Done THEN
				eInShutterAct	:= PneuActIdle;

				tyP0921InletNOutletShutter.tyInletShutterFB.tyBtnOpen.bValue	:= FALSE;
			ELSIF p_eInShutterStatus = Error THEN
				tyP0921InletNOutletShutter.tyInletShutterFB.tyBtnOpen.bValue	:= FALSE;
			END_IF

		ELSIF tyP0921InletNOutletShutter.tyInletShutterFB.tyBtnClose.bValue = TRUE THEN
			eInShutterAct	:= PneuActExt;

			IF p_eInShutterStat = PneuActExt AND p_eInShutterStatus = Done THEN
				eInShutterAct	:= PneuActIdle;

				tyP0921InletNOutletShutter.tyInletShutterFB.tyBtnClose.bValue := FALSE;
			ELSIF p_eInShutterStatus = Error THEN
				tyP0921InletNOutletShutter.tyInletShutterFB.tyBtnClose.bValue := FALSE;
			END_IF
		END_IF

		//Update Direct Control Status
		tyP0921InletNOutletShutter.tyInletShutterDC.tyBtnOpen.bRtCompl	:= FALSE;
		tyP0921InletNOutletShutter.tyInletShutterDC.tyBtnClose.bRtCompl	:= FALSE;
		tyP0921InletNOutletShutter.tyInletShutterDC.tyBtnOpen.bValue	:= p_bInShutterRetCtrl;
		tyP0921InletNOutletShutter.tyInletShutterDC.tyBtnClose.bValue	:= p_bInShutterExtCtrl;

	END_IF

END_ACTION
```

#### Act_OptP0921InletShutterFBStat.st
```iecst
ACTION Act_OptP0921InletShutterFBStat:

	tyP0921InletNOutletShutter.tyInletShutterFB.tyStringStat.sValue	:= p_sInShutterStatTxt;

END_ACTION
```

#### Act_OptP0921InletShutterDC.st
```iecst
ACTION Act_OptP0921InletShutterDC:

	IF tyP0921InletNOutletShutter.tyInletShutterCom.tyBtnSwitch.bValue = TRUE THEN
		IF p_bInShutterTwoCtrlOut = FALSE THEN
			IF tyP0921InletNOutletShutter.tyInletShutterDC.tyBtnOpen.bRtCompl = TRUE THEN
				tyP0921InletNOutletShutter.tyInletShutterDC.tyBtnOpen.bValue	:= TRUE;
				tyP0921InletNOutletShutter.tyInletShutterDC.tyBtnClose.bValue	:= FALSE;

				eInShutterAct	:= PneuActSetRet;

				IF p_eInShutterStat = PneuActSetRet AND p_eInShutterStatus = Done THEN
					eInShutterAct	:= PneuActIdle;

					tyP0921InletNOutletShutter.tyInletShutterDC.tyBtnOpen.bRtCompl	:= FALSE;
				END_IF

			ELSIF tyP0921InletNOutletShutter.tyInletShutterDC.tyBtnClose.bRtCompl = TRUE THEN
				tyP0921InletNOutletShutter.tyInletShutterDC.tyBtnClose.bValue	:= TRUE;
				tyP0921InletNOutletShutter.tyInletShutterDC.tyBtnOpen.bValue	:= FALSE;

				eInShutterAct	:= PneuActSetExt;

				IF p_eInShutterStat = PneuActSetExt AND p_eInShutterStatus = Done THEN
					eInShutterAct	:= PneuActIdle;

					tyP0921InletNOutletShutter.tyInletShutterDC.tyBtnClose.bRtCompl	:= FALSE;
				END_IF
			END_IF

		ELSE
			IF (tyP0921InletNOutletShutter.tyInletShutterDC.tyBtnOpen.bRtCompl = TRUE) OR (tyP0921InletNOutletShutter.tyInletShutterDC.tyBtnClose.bRtCompl = TRUE) THEN
				IF (tyP0921InletNOutletShutter.tyInletShutterDC.tyBtnOpen.bValue = TRUE) AND (tyP0921InletNOutletShutter.tyInletShutterDC.tyBtnClose.bValue = TRUE) THEN
					eInShutterAct	:= PneuActSetAll;

					IF p_eInShutterStat = PneuActSetAll AND p_eInShutterStatus = Done THEN
						eInShutterAct	:= PneuActIdle;

						tyP0921InletNOutletShutter.tyInletShutterDC.tyBtnOpen.bRtCompl	:= FALSE;
						tyP0921InletNOutletShutter.tyInletShutterDC.tyBtnClose.bRtCompl	:= FALSE;
					END_IF

				ELSIF (tyP0921InletNOutletShutter.tyInletShutterDC.tyBtnOpen.bValue = TRUE) AND (tyP0921InletNOutletShutter.tyInletShutterDC.tyBtnClose.bValue = FALSE) THEN
					eInShutterAct	:= PneuActSetRet;

					IF p_eInShutterStat = PneuActSetRet AND p_eInShutterStatus = Done THEN
						eInShutterAct	:= PneuActIdle;

						tyP0921InletNOutletShutter.tyInletShutterDC.tyBtnOpen.bRtCompl	:= FALSE;
						tyP0921InletNOutletShutter.tyInletShutterDC.tyBtnClose.bRtCompl	:= FALSE;
					END_IF

				ELSIF (tyP0921InletNOutletShutter.tyInletShutterDC.tyBtnOpen.bValue = FALSE) AND (tyP0921InletNOutletShutter.tyInletShutterDC.tyBtnClose.bValue = TRUE) THEN
					eInShutterAct	:= PneuActSetExt;

					IF p_eInShutterStat = PneuActSetExt AND p_eInShutterStatus = Done THEN
						eInShutterAct	:= PneuActIdle;

						tyP0921InletNOutletShutter.tyInletShutterDC.tyBtnOpen.bRtCompl	:= FALSE;
						tyP0921InletNOutletShutter.tyInletShutterDC.tyBtnClose.bRtCompl	:= FALSE;
					END_IF

				ELSE
					eInShutterAct	:= PneuActRstAll;

					IF p_eInShutterStat = PneuActRstAll AND p_eInShutterStatus = Done THEN
						eInShutterAct	:= PneuActIdle;

						tyP0921InletNOutletShutter.tyInletShutterDC.tyBtnOpen.bRtCompl	:= FALSE;
						tyP0921InletNOutletShutter.tyInletShutterDC.tyBtnClose.bRtCompl	:= FALSE;
					END_IF

				END_IF
			END_IF
		END_IF

		tyP0921InletNOutletShutter.tyInletShutterFB.tyBtnClose.bRtCompl	:= FALSE;
		tyP0921InletNOutletShutter.tyInletShutterFB.tyBtnClose.bValue	:= FALSE;
		tyP0921InletNOutletShutter.tyInletShutterFB.tyBtnOpen.bRtCompl	:= FALSE;
		tyP0921InletNOutletShutter.tyInletShutterFB.tyBtnOpen.bValue	:= FALSE;

	END_IF

END_ACTION
```

#### Act_OptP0921OutletShutterChgLyr.st
```iecst
ACTION Act_OptP0921OutletShutterChgLyr:

	IF	tyP0921InletNOutletShutter.tyOutletShutterCom.tyBtnSwitch.bRtCompl THEN
			tyP0921InletNOutletShutter.tyOutletShutterCom.tyBtnSwitch.bRtCompl := FALSE;

		IF tyP0921InletNOutletShutter.tyOutletShutterCom.tyBtnSwitch.bValue = TRUE THEN
			fUIInRtStatOff(ADR(tyP0921InletNOutletShutter.tyOutletShutterDC.tyLyr.uiRtStat));
			fUIInRtStatHide(ADR(tyP0921InletNOutletShutter.tyOutletShutterFB.tyLyr.uiRtStat));
		ELSE
			fUIInRtStatHide(ADR(tyP0921InletNOutletShutter.tyOutletShutterDC.tyLyr.uiRtStat));
			fUIInRtStatOff(ADR(tyP0921InletNOutletShutter.tyOutletShutterFB.tyLyr.uiRtStat));
		END_IF

	END_IF

END_ACTION
```

#### Act_OptP0921OutletShutterSen.st
```iecst
ACTION Act_OptP0921OutletShutterSen:

	tyP0921InletNOutletShutter.tyOutletShutterCom.tyBtnOpenRS.bValue	:= p_tyDI.bOutShutterOpenRS;
	tyP0921InletNOutletShutter.tyOutletShutterCom.tyBtnCloseRS.bValue	:= p_tyDI.bOutShutterCloseRS;

	//Machine Bitmap
	IF p_tyDI.bOutShutterOpenRS = TRUE THEN
		tyP0921InletNOutletShutter.tyOutletShutterCom.tyBitmapMc.uiValueIdx	:= 1;
	ELSE
		tyP0921InletNOutletShutter.tyOutletShutterCom.tyBitmapMc.uiValueIdx	:= 0;
	END_IF

	IF p_tyNtParamCurr.eProjMag = ULMagTriple THEN
		IF p_tyNtParamCurr.bProjLifterMagPlatform AND p_tyNtParamCurr.bUIConvDirRL THEN
			IF 	tyP0921InletNOutletShutter.tyOutletShutterCom.tyBitmapMc.uiValueIdx < 100 THEN
				tyP0921InletNOutletShutter.tyOutletShutterCom.tyBitmapMc.uiValueIdx	:= tyP0921InletNOutletShutter.tyOutletShutterCom.tyBitmapMc.uiValueIdx + 800;
			END_IF
		ELSIF p_tyNtParamCurr.bProjLifterMagPlatform THEN
			IF 	tyP0921InletNOutletShutter.tyOutletShutterCom.tyBitmapMc.uiValueIdx < 100 THEN
				tyP0921InletNOutletShutter.tyOutletShutterCom.tyBitmapMc.uiValueIdx	:= tyP0921InletNOutletShutter.tyOutletShutterCom.tyBitmapMc.uiValueIdx + 500;
				END_IF
		ELSIF p_tyNtParamCurr.bProjMagAWPrep = FALSE AND p_tyNtParamCurr.bProjMagSafetyBarPrep = FALSE THEN
			IF 	tyP0921InletNOutletShutter.tyOutletShutterCom.tyBitmapMc.uiValueIdx < 100 AND p_tyNtParamCurr.bCurtainSenPrep THEN

					tyP0921InletNOutletShutter.tyOutletShutterCom.tyBitmapMc.uiValueIdx	:= tyP0921InletNOutletShutter.tyOutletShutterCom.tyBitmapMc.uiValueIdx + 147;
			ELSE
					tyP0921InletNOutletShutter.tyOutletShutterCom.tyBitmapMc.uiValueIdx	:= tyP0921InletNOutletShutter.tyOutletShutterCom.tyBitmapMc.uiValueIdx + 100;
			END_IF
		ELSIF p_tyNtParamCurr.eProjMag = ULMagTriple AND p_tyNtParamCurr.bProjMagAWPrep THEN
			IF 	tyP0921InletNOutletShutter.tyOutletShutterCom.tyBitmapMc.uiValueIdx < 134 THEN
				tyP0921InletNOutletShutter.tyOutletShutterCom.tyBitmapMc.uiValueIdx	:= tyP0921InletNOutletShutter.tyOutletShutterCom.tyBitmapMc.uiValueIdx + 134;
			END_IF
		ELSIF p_tyNtParamCurr.bProjMagAWPrep = FALSE AND p_tyNtParamCurr.bProjMagSafetyBarPrep = TRUE THEN
			IF 	tyP0921InletNOutletShutter.tyOutletShutterCom.tyBitmapMc.uiValueIdx < 402 THEN
				tyP0921InletNOutletShutter.tyOutletShutterCom.tyBitmapMc.uiValueIdx	:= tyP0921InletNOutletShutter.tyOutletShutterCom.tyBitmapMc.uiValueIdx + 402;
			END_IF
		END_IF
	ELSIF p_tyNtParamCurr.eProjMag = ULMagDual THEN
		IF p_tyNtParamCurr.bProjLifterMagPlatform AND p_tyNtParamCurr.bUIConvDirRL THEN
			IF 	tyP0921InletNOutletShutter.tyOutletShutterCom.tyBitmapMc.uiValueIdx < 100 THEN
				tyP0921InletNOutletShutter.tyOutletShutterCom.tyBitmapMc.uiValueIdx	:= tyP0921InletNOutletShutter.tyOutletShutterCom.tyBitmapMc.uiValueIdx + 700;
			END_IF
		ELSIF p_tyNtParamCurr.bProjLifterMagPlatform AND p_tyNtParamCurr.bUIConvDirRL = FALSE AND p_tyNtParamCurr.bProjMagConvLane1Prep THEN
			IF 	tyP0921InletNOutletShutter.tyOutletShutterCom.tyBitmapMc.uiValueIdx < 100 THEN
				tyP0921InletNOutletShutter.tyOutletShutterCom.tyBitmapMc.uiValueIdx	:= tyP0921InletNOutletShutter.tyOutletShutterCom.tyBitmapMc.uiValueIdx + 900;
			END_IF
		ELSIF p_tyNtParamCurr.bProjLifterMagPlatform THEN
				IF 	tyP0921InletNOutletShutter.tyOutletShutterCom.tyBitmapMc.uiValueIdx < 100 THEN
					tyP0921InletNOutletShutter.tyOutletShutterCom.tyBitmapMc.uiValueIdx	:= tyP0921InletNOutletShutter.tyOutletShutterCom.tyBitmapMc.uiValueIdx + 600;
				END_IF
		ELSIF p_tyNtParamCurr.bProjMagAWPrep = FALSE THEN
			tyP0921InletNOutletShutter.tyOutletShutterCom.tyBitmapMc.uiValueIdx	:= tyP0921InletNOutletShutter.tyOutletShutterCom.tyBitmapMc.uiValueIdx + 3;
		ELSIF p_tyNtParamCurr.bProjMagAWPrep THEN
			tyP0921InletNOutletShutter.tyOutletShutterCom.tyBitmapMc.uiValueIdx	:= tyP0921InletNOutletShutter.tyOutletShutterCom.tyBitmapMc.uiValueIdx + 334;
		END_IF
	END_IF

END_ACTION
```

#### Act_OptP0921OutletShutterFB.st
```iecst
ACTION Act_OptP0921OutletShutterFB:

	IF tyP0921InletNOutletShutter.tyOutletShutterCom.tyBtnSwitch.bValue = FALSE THEN
		// FB Control
		IF tyP0921InletNOutletShutter.tyOutletShutterFB.tyBtnOpen.bRtCompl = TRUE THEN
			tyP0921InletNOutletShutter.tyOutletShutterFB.tyBtnOpen.bRtCompl	:= FALSE;

			tyP0921InletNOutletShutter.tyOutletShutterFB.tyBtnOpen.bValue	:= TRUE;
			tyP0921InletNOutletShutter.tyOutletShutterFB.tyBtnClose.bValue	:= FALSE;

		ELSIF tyP0921InletNOutletShutter.tyOutletShutterFB.tyBtnClose.bRtCompl = TRUE THEN
			tyP0921InletNOutletShutter.tyOutletShutterFB.tyBtnClose.bRtCompl	:= FALSE;

			tyP0921InletNOutletShutter.tyOutletShutterFB.tyBtnClose.bValue	:= TRUE;
			tyP0921InletNOutletShutter.tyOutletShutterFB.tyBtnOpen.bValue	:= FALSE;
		END_IF

		IF tyP0921InletNOutletShutter.tyOutletShutterFB.tyBtnOpen.bValue = TRUE THEN
			eOutShutterAct	:= PneuActRet;

			IF p_eOutShutterStat = PneuActRet AND p_eOutShutterStatus = Done THEN
				eOutShutterAct	:= PneuActIdle;

				tyP0921InletNOutletShutter.tyOutletShutterFB.tyBtnOpen.bValue	:= FALSE;
			ELSIF p_eOutShutterStatus = Error THEN
				tyP0921InletNOutletShutter.tyOutletShutterFB.tyBtnOpen.bValue	:= FALSE;
			END_IF

		ELSIF tyP0921InletNOutletShutter.tyOutletShutterFB.tyBtnClose.bValue = TRUE THEN
			eOutShutterAct		:= PneuActExt;

			IF p_eOutShutterStat = PneuActExt AND p_eOutShutterStatus = Done THEN

				eOutShutterAct	:= PneuActIdle;

				tyP0921InletNOutletShutter.tyOutletShutterFB.tyBtnClose.bValue := FALSE;
			ELSIF p_eOutShutterStatus = Error THEN
				tyP0921InletNOutletShutter.tyOutletShutterFB.tyBtnClose.bValue := FALSE;
			END_IF

		END_IF

		//UpdateStatus
		tyP0921InletNOutletShutter.tyOutletShutterDC.tyBtnClose.bRtCompl	:= FALSE;
		tyP0921InletNOutletShutter.tyOutletShutterDC.tyBtnOpen.bRtCompl		:= FALSE;
		tyP0921InletNOutletShutter.tyOutletShutterDC.tyBtnClose.bValue		:= p_bOutShutterExtCtrl;
		tyP0921InletNOutletShutter.tyOutletShutterDC.tyBtnOpen.bValue		:= p_bOutShutterRetCtrl;

	END_IF

END_ACTION
```

#### Act_OptP0921OutletShutterFBStat.st
```iecst
ACTION Act_OptP0921OutletShutterFBStat:

	tyP0921InletNOutletShutter.tyOutletShutterFB.tyStringStat.sValue	:= p_sOutShutterStatTxt;

END_ACTION
```

#### Act_OptP0921OutletShutterDC.st
```iecst
ACTION Act_OptP0921OutletShutterDC:

	// Direct Control
	IF tyP0921InletNOutletShutter.tyOutletShutterCom.tyBtnSwitch.bValue = TRUE THEN
		IF p_bOutShutterTwoCtrlOut = FALSE THEN
			IF tyP0921InletNOutletShutter.tyOutletShutterDC.tyBtnOpen.bRtCompl = TRUE THEN
				tyP0921InletNOutletShutter.tyOutletShutterDC.tyBtnOpen.bValue	:= TRUE;
				tyP0921InletNOutletShutter.tyOutletShutterDC.tyBtnClose.bValue	:= FALSE;

				eOutShutterAct	:= PneuActSetRet;

				IF p_eOutShutterStat = PneuActSetRet AND p_eOutShutterStatus = Done THEN
					eOutShutterAct	:= PneuActIdle;

					tyP0921InletNOutletShutter.tyOutletShutterDC.tyBtnOpen.bRtCompl	:= FALSE;
				END_IF

			ELSIF tyP0921InletNOutletShutter.tyOutletShutterDC.tyBtnClose.bRtCompl = TRUE THEN
				tyP0921InletNOutletShutter.tyOutletShutterDC.tyBtnClose.bValue	:= TRUE;
				tyP0921InletNOutletShutter.tyOutletShutterDC.tyBtnOpen.bValue	:= FALSE;

				eOutShutterAct	:= PneuActSetExt;

				IF p_eOutShutterStat = PneuActSetExt AND p_eOutShutterStatus = Done THEN
					eOutShutterAct	:= PneuActIdle;

					tyP0921InletNOutletShutter.tyOutletShutterDC.tyBtnClose.bRtCompl	:= FALSE;
				END_IF
			END_IF

		ELSE
			IF (tyP0921InletNOutletShutter.tyOutletShutterDC.tyBtnOpen.bRtCompl = TRUE) OR (tyP0921InletNOutletShutter.tyOutletShutterDC.tyBtnClose.bRtCompl = TRUE) THEN
				IF (tyP0921InletNOutletShutter.tyOutletShutterDC.tyBtnOpen.bValue = TRUE) AND (tyP0921InletNOutletShutter.tyOutletShutterDC.tyBtnClose.bValue = TRUE) THEN
					eOutShutterAct	:= PneuActSetAll;

					IF p_eOutShutterStat = PneuActSetAll AND p_eOutShutterStatus = Done THEN
						eOutShutterAct	:= PneuActIdle;

						tyP0921InletNOutletShutter.tyOutletShutterDC.tyBtnOpen.bRtCompl		:= FALSE;
						tyP0921InletNOutletShutter.tyOutletShutterDC.tyBtnClose.bRtCompl	:= FALSE;
					END_IF

				ELSIF (tyP0921InletNOutletShutter.tyOutletShutterDC.tyBtnOpen.bValue = TRUE) AND (tyP0921InletNOutletShutter.tyOutletShutterDC.tyBtnClose.bValue = FALSE) THEN
					eOutShutterAct	:= PneuActSetRet;

					IF p_eOutShutterStat = PneuActSetRet AND p_eOutShutterStatus = Done THEN
						eOutShutterAct	:= PneuActIdle;

						tyP0921InletNOutletShutter.tyOutletShutterDC.tyBtnOpen.bRtCompl		:= FALSE;
						tyP0921InletNOutletShutter.tyOutletShutterDC.tyBtnClose.bRtCompl	:= FALSE;
					END_IF

				ELSIF (tyP0921InletNOutletShutter.tyOutletShutterDC.tyBtnOpen.bValue = FALSE) AND (tyP0921InletNOutletShutter.tyOutletShutterDC.tyBtnClose.bValue = TRUE) THEN
					eOutShutterAct	:= PneuActSetExt;

					IF p_eOutShutterStat = PneuActSetExt AND p_eOutShutterStatus = Done THEN
						eOutShutterAct	:= PneuActIdle;

						tyP0921InletNOutletShutter.tyOutletShutterDC.tyBtnOpen.bRtCompl		:= FALSE;
						tyP0921InletNOutletShutter.tyOutletShutterDC.tyBtnClose.bRtCompl	:= FALSE;
					END_IF

				ELSE
					eOutShutterAct	:= PneuActRstAll;

					IF p_eOutShutterStat = PneuActRstAll AND p_eOutShutterStatus = Done THEN
						eOutShutterAct	:= PneuActIdle;

						tyP0921InletNOutletShutter.tyOutletShutterDC.tyBtnOpen.bRtCompl		:= FALSE;
						tyP0921InletNOutletShutter.tyOutletShutterDC.tyBtnClose.bRtCompl	:= FALSE;
					END_IF

				END_IF
			END_IF
		END_IF

		tyP0921InletNOutletShutter.tyOutletShutterFB.tyBtnOpen.bRtCompl	:= FALSE;
		tyP0921InletNOutletShutter.tyOutletShutterFB.tyBtnOpen.bValue	:= FALSE;
		tyP0921InletNOutletShutter.tyOutletShutterFB.tyBtnClose.bRtCompl:= FALSE;
		tyP0921InletNOutletShutter.tyOutletShutterFB.tyBtnClose.bValue	:= FALSE;

	END_IF

END_ACTION
```

#### Act_OptP0921RstMnl.st
```iecst
ACTION Act_OptP0921RstMnl:

	IF EDGEPOS((bManualMod = FALSE) OR (p_eInShutterStatus = Error)) THEN

		eInShutterAct	:= PneuActIdle;

		tyP0921InletNOutletShutter.tyInletShutterDC.tyBtnClose.bRtCompl	:= FALSE;
		tyP0921InletNOutletShutter.tyInletShutterDC.tyBtnClose.bValue	:= FALSE;
		tyP0921InletNOutletShutter.tyInletShutterDC.tyBtnOpen.bRtCompl	:= FALSE;
		tyP0921InletNOutletShutter.tyInletShutterDC.tyBtnOpen.bValue	:= TRUE;

		tyP0921InletNOutletShutter.tyInletShutterFB.tyBtnClose.bRtCompl	:= FALSE;
		tyP0921InletNOutletShutter.tyInletShutterFB.tyBtnClose.bValue	:= FALSE;
		tyP0921InletNOutletShutter.tyInletShutterFB.tyBtnOpen.bRtCompl	:= FALSE;
		tyP0921InletNOutletShutter.tyInletShutterFB.tyBtnOpen.bValue	:= FALSE;

	END_IF

	IF EDGEPOS((bManualMod = FALSE) OR (p_eOutShutterStatus = Error)) THEN

		eOutShutterAct	:= PneuActIdle;

		tyP0921InletNOutletShutter.tyOutletShutterDC.tyBtnClose.bRtCompl	:= FALSE;
		tyP0921InletNOutletShutter.tyOutletShutterDC.tyBtnClose.bValue		:= FALSE;
		tyP0921InletNOutletShutter.tyOutletShutterDC.tyBtnOpen.bRtCompl		:= FALSE;
		tyP0921InletNOutletShutter.tyOutletShutterDC.tyBtnOpen.bValue		:= FALSE;

		tyP0921InletNOutletShutter.tyOutletShutterFB.tyBtnClose.bRtCompl	:= FALSE;
		tyP0921InletNOutletShutter.tyOutletShutterFB.tyBtnClose.bValue		:= FALSE;
		tyP0921InletNOutletShutter.tyOutletShutterFB.tyBtnOpen.bRtCompl		:= FALSE;
		tyP0921InletNOutletShutter.tyOutletShutterFB.tyBtnOpen.bValue		:= FALSE;

	END_IF

	IF EDGEPOS(bManualMod = FALSE) THEN
		tyP0921InletNOutletShutter.tyInletShutterCom.tyBtnSwitch.bValue := FALSE;
		tyP0921InletNOutletShutter.tyOutletShutterCom.tyBtnSwitch.bValue := FALSE;

		IF p_tyNtParamCurr.bProjInletShutPrep THEN
			fUIInRtStatHide(ADR(tyP0921InletNOutletShutter.tyInletShutterDC.tyLyr.uiRtStat));
			fUIInRtStatOff(ADR(tyP0921InletNOutletShutter.tyInletShutterFB.tyLyr.uiRtStat));
		ELSE
			fUIInRtStatHide(ADR(tyP0921InletNOutletShutter.tyInletShutterFB.tyLyr.uiRtStat));
		END_IF
		IF p_tyNtParamCurr.bProjOutletShutPrep THEN
			fUIInRtStatHide(ADR(tyP0921InletNOutletShutter.tyOutletShutterDC.tyLyr.uiRtStat));
			fUIInRtStatOff(ADR(tyP0921InletNOutletShutter.tyOutletShutterFB.tyLyr.uiRtStat));
		ELSE
			fUIInRtStatHide(ADR(tyP0921InletNOutletShutter.tyOutletShutterFB.tyLyr.uiRtStat));
		END_IF

	END_IF

END_ACTION
```

#### Act_OptP0921OutletShutterChgLyr3.st
```iecst
ACTION Act_OptP0921OutletShutterChgLyr3:

	IF	tyP0921InletNOutletShutter.tyOutletShutterCom3.tyBtnSwitch.bRtCompl THEN
			tyP0921InletNOutletShutter.tyOutletShutterCom3.tyBtnSwitch.bRtCompl := FALSE;

		IF tyP0921InletNOutletShutter.tyOutletShutterCom3.tyBtnSwitch.bValue = TRUE THEN
			fUIInRtStatOff(ADR(tyP0921InletNOutletShutter.tyOutletShutterDC3.tyLyr.uiRtStat));
			fUIInRtStatHide(ADR(tyP0921InletNOutletShutter.tyOutletShutterFB3.tyLyr.uiRtStat));
		ELSE
			fUIInRtStatHide(ADR(tyP0921InletNOutletShutter.tyOutletShutterDC3.tyLyr.uiRtStat));
			fUIInRtStatOff(ADR(tyP0921InletNOutletShutter.tyOutletShutterFB3.tyLyr.uiRtStat));
		END_IF

	END_IF

END_ACTION
```

#### Act_OptP0921OutletShutterSen3.st
```iecst
ACTION Act_OptP0921OutletShutterSen3:

	tyP0921InletNOutletShutter.tyOutletShutterCom3.tyBtnOpenRS.bValue	:= p_tyDI.bOutShutterOpenRS3;
	tyP0921InletNOutletShutter.tyOutletShutterCom3.tyBtnCloseRS.bValue	:= p_tyDI.bOutShutterCloseRS3;

	//Machine Bitmap
	IF p_tyDI.bOutShutterOpenRS3 = TRUE THEN
		tyP0921InletNOutletShutter.tyOutletShutterCom3.tyBitmapMc.uiValueIdx	:= 1;
	ELSE
		tyP0921InletNOutletShutter.tyOutletShutterCom3.tyBitmapMc.uiValueIdx	:= 0;

	END_IF

	IF p_tyNtParamCurr.eProjMag = ULMagTriple THEN
		IF p_tyNtParamCurr.bProjLifterMagPlatform AND p_tyNtParamCurr.bUIConvDirRL THEN
			IF 	tyP0921InletNOutletShutter.tyOutletShutterCom3.tyBitmapMc.uiValueIdx < 100 THEN
				tyP0921InletNOutletShutter.tyOutletShutterCom3.tyBitmapMc.uiValueIdx	:= tyP0921InletNOutletShutter.tyOutletShutterCom3.tyBitmapMc.uiValueIdx + 800;
			END_IF
		ELSIF p_tyNtParamCurr.bProjLifterMagPlatform THEN
			IF 	tyP0921InletNOutletShutter.tyOutletShutterCom3.tyBitmapMc.uiValueIdx < 100 THEN
				tyP0921InletNOutletShutter.tyOutletShutterCom3.tyBitmapMc.uiValueIdx	:= tyP0921InletNOutletShutter.tyOutletShutterCom3.tyBitmapMc.uiValueIdx + 500;
				END_IF
		ELSIF p_tyNtParamCurr.bProjMagAWPrep = FALSE AND p_tyNtParamCurr.bProjMagSafetyBarPrep = FALSE THEN
			IF 	tyP0921InletNOutletShutter.tyOutletShutterCom3.tyBitmapMc.uiValueIdx < 100 AND  p_tyNtParamCurr.bCurtainSenPrep THEN

				tyP0921InletNOutletShutter.tyOutletShutterCom3.tyBitmapMc.uiValueIdx	:= tyP0921InletNOutletShutter.tyOutletShutterCom3.tyBitmapMc.uiValueIdx + 151;
			ELSE
				tyP0921InletNOutletShutter.tyOutletShutterCom3.tyBitmapMc.uiValueIdx	:= tyP0921InletNOutletShutter.tyOutletShutterCom3.tyBitmapMc.uiValueIdx + 100;

			END_IF
		ELSIF p_tyNtParamCurr.eProjMag = ULMagTriple AND p_tyNtParamCurr.bProjMagAWPrep THEN
			IF 	tyP0921InletNOutletShutter.tyOutletShutterCom3.tyBitmapMc.uiValueIdx < 134 THEN
				tyP0921InletNOutletShutter.tyOutletShutterCom3.tyBitmapMc.uiValueIdx	:= tyP0921InletNOutletShutter.tyOutletShutterCom3.tyBitmapMc.uiValueIdx + 134;
			END_IF
		ELSIF p_tyNtParamCurr.bProjMagAWPrep = FALSE AND p_tyNtParamCurr.bProjMagSafetyBarPrep = TRUE THEN
			IF 	tyP0921InletNOutletShutter.tyOutletShutterCom3.tyBitmapMc.uiValueIdx < 402 THEN
				tyP0921InletNOutletShutter.tyOutletShutterCom3.tyBitmapMc.uiValueIdx	:= tyP0921InletNOutletShutter.tyOutletShutterCom3.tyBitmapMc.uiValueIdx + 400;
			END_IF
		END_IF
	ELSIF p_tyNtParamCurr.eProjMag = ULMagDual THEN
		IF p_tyNtParamCurr.bProjLifterMagPlatform AND p_tyNtParamCurr.bUIConvDirRL THEN
			IF 	tyP0921InletNOutletShutter.tyOutletShutterCom3.tyBitmapMc.uiValueIdx < 100 THEN
				tyP0921InletNOutletShutter.tyOutletShutterCom3.tyBitmapMc.uiValueIdx	:= tyP0921InletNOutletShutter.tyOutletShutterCom3.tyBitmapMc.uiValueIdx + 700;
			END_IF
		ELSIF p_tyNtParamCurr.bProjLifterMagPlatform AND p_tyNtParamCurr.bUIConvDirRL = FALSE AND p_tyNtParamCurr.bProjMagConvLane1Prep THEN
			IF 	tyP0921InletNOutletShutter.tyOutletShutterCom3.tyBitmapMc.uiValueIdx < 100 THEN
				tyP0921InletNOutletShutter.tyOutletShutterCom3.tyBitmapMc.uiValueIdx	:= tyP0921InletNOutletShutter.tyOutletShutterCom3.tyBitmapMc.uiValueIdx + 900;
			END_IF
		ELSIF p_tyNtParamCurr.bProjLifterMagPlatform THEN
				IF 	tyP0921InletNOutletShutter.tyOutletShutterCom3.tyBitmapMc.uiValueIdx < 100 THEN
					tyP0921InletNOutletShutter.tyOutletShutterCom3.tyBitmapMc.uiValueIdx	:= tyP0921InletNOutletShutter.tyOutletShutterCom3.tyBitmapMc.uiValueIdx + 600;
				END_IF
		ELSIF p_tyNtParamCurr.bProjMagAWPrep = FALSE THEN
			tyP0921InletNOutletShutter.tyOutletShutterCom3.tyBitmapMc.uiValueIdx	:= tyP0921InletNOutletShutter.tyOutletShutterCom3.tyBitmapMc.uiValueIdx + 3;
		ELSIF p_tyNtParamCurr.bProjMagAWPrep THEN
			tyP0921InletNOutletShutter.tyOutletShutterCom3.tyBitmapMc.uiValueIdx	:= tyP0921InletNOutletShutter.tyOutletShutterCom3.tyBitmapMc.uiValueIdx + 334;
		END_IF
	END_IF

END_ACTION
```

#### Act_OptP0921OutletShutterFB3.st
```iecst
ACTION Act_OptP0921OutletShutterFB3:

	IF tyP0921InletNOutletShutter.tyOutletShutterCom3.tyBtnSwitch.bValue = FALSE THEN
		// FB Control
		IF tyP0921InletNOutletShutter.tyOutletShutterFB3.tyBtnOpen.bRtCompl = TRUE THEN
			tyP0921InletNOutletShutter.tyOutletShutterFB3.tyBtnOpen.bRtCompl	:= FALSE;

			tyP0921InletNOutletShutter.tyOutletShutterFB3.tyBtnOpen.bValue	:= TRUE;
			tyP0921InletNOutletShutter.tyOutletShutterFB3.tyBtnClose.bValue	:= FALSE;

		ELSIF tyP0921InletNOutletShutter.tyOutletShutterFB3.tyBtnClose.bRtCompl = TRUE THEN
			tyP0921InletNOutletShutter.tyOutletShutterFB3.tyBtnClose.bRtCompl	:= FALSE;

			tyP0921InletNOutletShutter.tyOutletShutterFB3.tyBtnClose.bValue	:= TRUE;
			tyP0921InletNOutletShutter.tyOutletShutterFB3.tyBtnOpen.bValue	:= FALSE;
		END_IF

		IF tyP0921InletNOutletShutter.tyOutletShutterFB3.tyBtnOpen.bValue = TRUE THEN
			eOutShutterAct3	:= PneuActRet;

			IF p_eOutShutterStat3 = PneuActRet AND p_eOutShutterStatus3 = Done THEN
				eOutShutterAct3	:= PneuActIdle;

				tyP0921InletNOutletShutter.tyOutletShutterFB3.tyBtnOpen.bValue	:= FALSE;
			ELSIF p_eOutShutterStatus3 = Error THEN
				tyP0921InletNOutletShutter.tyOutletShutterFB3.tyBtnOpen.bValue	:= FALSE;
			END_IF

		ELSIF tyP0921InletNOutletShutter.tyOutletShutterFB3.tyBtnClose.bValue = TRUE THEN
			eOutShutterAct3		:= PneuActExt;

			IF p_eOutShutterStat3 = PneuActExt AND p_eOutShutterStatus3 = Done THEN

				eOutShutterAct3	:= PneuActIdle;

				tyP0921InletNOutletShutter.tyOutletShutterFB3.tyBtnClose.bValue := FALSE;
			ELSIF p_eOutShutterStatus3 = Error THEN
				tyP0921InletNOutletShutter.tyOutletShutterFB3.tyBtnClose.bValue := FALSE;
			END_IF

		END_IF

		//UpdateStatus
		tyP0921InletNOutletShutter.tyOutletShutterDC3.tyBtnClose.bRtCompl		:= FALSE;
		tyP0921InletNOutletShutter.tyOutletShutterDC3.tyBtnOpen.bRtCompl		:= FALSE;
		tyP0921InletNOutletShutter.tyOutletShutterDC3.tyBtnClose.bValue			:= p_bOutShutterExtCtrl3;
		tyP0921InletNOutletShutter.tyOutletShutterDC3.tyBtnOpen.bValue			:= p_bOutShutterRetCtrl3;

	END_IF

END_ACTION
```

#### Act_OptP0921OutletShutterFBStat3.st
```iecst
ACTION Act_OptP0921OutletShutterFBStat3:

	tyP0921InletNOutletShutter.tyOutletShutterFB3.tyStringStat.sValue	:= p_sOutShutterStatTxt3;

END_ACTION
```

#### Act_OptP0921OutletShutterDC3.st
```iecst
ACTION Act_OptP0921OutletShutterDC3:

	// Direct Control
	IF tyP0921InletNOutletShutter.tyOutletShutterCom3.tyBtnSwitch.bValue = TRUE THEN
		IF p_bOutShutterTwoCtrlOut3 = FALSE THEN
			IF tyP0921InletNOutletShutter.tyOutletShutterDC3.tyBtnOpen.bRtCompl = TRUE THEN
				tyP0921InletNOutletShutter.tyOutletShutterDC3.tyBtnOpen.bValue	:= TRUE;
				tyP0921InletNOutletShutter.tyOutletShutterDC3.tyBtnClose.bValue	:= FALSE;

				eOutShutterAct3	:= PneuActSetRet;

				IF p_eOutShutterStat3 = PneuActSetRet AND p_eOutShutterStatus3 = Done THEN
					eOutShutterAct3	:= PneuActIdle;

					tyP0921InletNOutletShutter.tyOutletShutterDC3.tyBtnOpen.bRtCompl	:= FALSE;
				END_IF

			ELSIF tyP0921InletNOutletShutter.tyOutletShutterDC3.tyBtnClose.bRtCompl = TRUE THEN
				tyP0921InletNOutletShutter.tyOutletShutterDC3.tyBtnClose.bValue	:= TRUE;
				tyP0921InletNOutletShutter.tyOutletShutterDC3.tyBtnOpen.bValue	:= FALSE;

				eOutShutterAct3	:= PneuActSetExt;

				IF p_eOutShutterStat3 = PneuActSetExt AND p_eOutShutterStatus3 = Done THEN
					eOutShutterAct3	:= PneuActIdle;

					tyP0921InletNOutletShutter.tyOutletShutterDC3.tyBtnClose.bRtCompl	:= FALSE;
				END_IF
			END_IF

		ELSE
			IF (tyP0921InletNOutletShutter.tyOutletShutterDC3.tyBtnOpen.bRtCompl = TRUE) OR (tyP0921InletNOutletShutter.tyOutletShutterDC3.tyBtnClose.bRtCompl = TRUE) THEN
				IF (tyP0921InletNOutletShutter.tyOutletShutterDC3.tyBtnOpen.bValue = TRUE) AND (tyP0921InletNOutletShutter.tyOutletShutterDC3.tyBtnClose.bValue = TRUE) THEN
					eOutShutterAct3	:= PneuActSetAll;

					IF p_eOutShutterStat3 = PneuActSetAll AND p_eOutShutterStatus3 = Done THEN
						eOutShutterAct3	:= PneuActIdle;

						tyP0921InletNOutletShutter.tyOutletShutterDC3.tyBtnOpen.bRtCompl		:= FALSE;
						tyP0921InletNOutletShutter.tyOutletShutterDC3.tyBtnClose.bRtCompl	:= FALSE;
					END_IF

				ELSIF (tyP0921InletNOutletShutter.tyOutletShutterDC3.tyBtnOpen.bValue = TRUE) AND (tyP0921InletNOutletShutter.tyOutletShutterDC3.tyBtnClose.bValue = FALSE) THEN
					eOutShutterAct3	:= PneuActSetRet;

					IF p_eOutShutterStat3 = PneuActSetRet AND p_eOutShutterStatus3 = Done THEN
						eOutShutterAct3	:= PneuActIdle;

						tyP0921InletNOutletShutter.tyOutletShutterDC3.tyBtnOpen.bRtCompl		:= FALSE;
						tyP0921InletNOutletShutter.tyOutletShutterDC3.tyBtnClose.bRtCompl	:= FALSE;
					END_IF

				ELSIF (tyP0921InletNOutletShutter.tyOutletShutterDC3.tyBtnOpen.bValue = FALSE) AND (tyP0921InletNOutletShutter.tyOutletShutterDC3.tyBtnClose.bValue = TRUE) THEN
					eOutShutterAct3	:= PneuActSetExt;

					IF p_eOutShutterStat3 = PneuActSetExt AND p_eOutShutterStatus3 = Done THEN
						eOutShutterAct3	:= PneuActIdle;

						tyP0921InletNOutletShutter.tyOutletShutterDC3.tyBtnOpen.bRtCompl		:= FALSE;
						tyP0921InletNOutletShutter.tyOutletShutterDC3.tyBtnClose.bRtCompl	:= FALSE;
					END_IF

				ELSE
					eOutShutterAct3	:= PneuActRstAll;

					IF p_eOutShutterStat3 = PneuActRstAll AND p_eOutShutterStatus3 = Done THEN
						eOutShutterAct3	:= PneuActIdle;

						tyP0921InletNOutletShutter.tyOutletShutterDC3.tyBtnOpen.bRtCompl		:= FALSE;
						tyP0921InletNOutletShutter.tyOutletShutterDC3.tyBtnClose.bRtCompl		:= FALSE;
					END_IF

				END_IF
			END_IF
		END_IF

		tyP0921InletNOutletShutter.tyOutletShutterFB3.tyBtnOpen.bRtCompl	:= FALSE;
		tyP0921InletNOutletShutter.tyOutletShutterFB3.tyBtnOpen.bValue		:= FALSE;
		tyP0921InletNOutletShutter.tyOutletShutterFB3.tyBtnClose.bRtCompl	:= FALSE;
		tyP0921InletNOutletShutter.tyOutletShutterFB3.tyBtnClose.bValue		:= FALSE;

	END_IF

END_ACTION
```

#### Act_OptP0921OutletShutterChgLyr2.st
```iecst
ACTION Act_OptP0921OutletShutterChgLyr2:

	IF	tyP0921InletNOutletShutter.tyOutletShutterCom2.tyBtnSwitch.bRtCompl THEN
			tyP0921InletNOutletShutter.tyOutletShutterCom2.tyBtnSwitch.bRtCompl := FALSE;

		IF tyP0921InletNOutletShutter.tyOutletShutterCom2.tyBtnSwitch.bValue = TRUE THEN
			fUIInRtStatOff(ADR(tyP0921InletNOutletShutter.tyOutletShutterDC2.tyLyr.uiRtStat));
			fUIInRtStatHide(ADR(tyP0921InletNOutletShutter.tyOutletShutterFB2.tyLyr.uiRtStat));
		ELSE
			fUIInRtStatHide(ADR(tyP0921InletNOutletShutter.tyOutletShutterDC2.tyLyr.uiRtStat));
			fUIInRtStatOff(ADR(tyP0921InletNOutletShutter.tyOutletShutterFB2.tyLyr.uiRtStat));
		END_IF

	END_IF

END_ACTION
```

#### Act_OptP0921OutletShutterSen2.st
```iecst
ACTION Act_OptP0921OutletShutterSen2:

	tyP0921InletNOutletShutter.tyOutletShutterCom2.tyBtnOpenRS.bValue	:= p_tyDI.bOutShutterOpenRS2;
	tyP0921InletNOutletShutter.tyOutletShutterCom2.tyBtnCloseRS.bValue	:= p_tyDI.bOutShutterCloseRS2;

	//Machine Bitmap
	IF p_tyDI.bOutShutterOpenRS2 = TRUE THEN
		tyP0921InletNOutletShutter.tyOutletShutterCom2.tyBitmapMc.uiValueIdx	:= 1;
	ELSE
		tyP0921InletNOutletShutter.tyOutletShutterCom2.tyBitmapMc.uiValueIdx	:= 0;
	END_IF

	IF p_tyNtParamCurr.eProjMag = ULMagTriple THEN
		IF p_tyNtParamCurr.bProjLifterMagPlatform AND p_tyNtParamCurr.bUIConvDirRL THEN
			IF 	tyP0921InletNOutletShutter.tyOutletShutterCom2.tyBitmapMc.uiValueIdx < 100 THEN
				tyP0921InletNOutletShutter.tyOutletShutterCom2.tyBitmapMc.uiValueIdx	:= tyP0921InletNOutletShutter.tyOutletShutterCom2.tyBitmapMc.uiValueIdx + 801;
			END_IF
		ELSIF p_tyNtParamCurr.bProjLifterMagPlatform THEN
			IF 	tyP0921InletNOutletShutter.tyOutletShutterCom2.tyBitmapMc.uiValueIdx < 100 THEN
				tyP0921InletNOutletShutter.tyOutletShutterCom2.tyBitmapMc.uiValueIdx	:= tyP0921InletNOutletShutter.tyOutletShutterCom2.tyBitmapMc.uiValueIdx + 501;
				END_IF
		ELSIF p_tyNtParamCurr.bProjMagAWPrep = FALSE AND p_tyNtParamCurr.bProjMagSafetyBarPrep = FALSE THEN
			IF 	tyP0921InletNOutletShutter.tyOutletShutterCom2.tyBitmapMc.uiValueIdx < 100 AND  p_tyNtParamCurr.bCurtainSenPrep THEN
					tyP0921InletNOutletShutter.tyOutletShutterCom2.tyBitmapMc.uiValueIdx	:= tyP0921InletNOutletShutter.tyOutletShutterCom2.tyBitmapMc.uiValueIdx + 151;
			ELSE
					tyP0921InletNOutletShutter.tyOutletShutterCom2.tyBitmapMc.uiValueIdx	:= tyP0921InletNOutletShutter.tyOutletShutterCom2.tyBitmapMc.uiValueIdx + 101;
			END_IF
		ELSIF p_tyNtParamCurr.eProjMag = ULMagTriple AND p_tyNtParamCurr.bProjMagAWPrep THEN
			IF 	tyP0921InletNOutletShutter.tyOutletShutterCom2.tyBitmapMc.uiValueIdx < 134 THEN
				tyP0921InletNOutletShutter.tyOutletShutterCom2.tyBitmapMc.uiValueIdx	:= tyP0921InletNOutletShutter.tyOutletShutterCom2.tyBitmapMc.uiValueIdx + 135;
			END_IF
		ELSIF p_tyNtParamCurr.bProjMagAWPrep = FALSE AND p_tyNtParamCurr.bProjMagSafetyBarPrep = TRUE THEN
			IF 	tyP0921InletNOutletShutter.tyOutletShutterCom2.tyBitmapMc.uiValueIdx < 402 THEN
				tyP0921InletNOutletShutter.tyOutletShutterCom2.tyBitmapMc.uiValueIdx	:= tyP0921InletNOutletShutter.tyOutletShutterCom2.tyBitmapMc.uiValueIdx + 403;
			END_IF
		END_IF
	ELSIF p_tyNtParamCurr.eProjMag = ULMagDual THEN
		IF p_tyNtParamCurr.bProjLifterMagPlatform AND p_tyNtParamCurr.bUIConvDirRL THEN
			IF 	tyP0921InletNOutletShutter.tyOutletShutterCom2.tyBitmapMc.uiValueIdx < 100 THEN
				tyP0921InletNOutletShutter.tyOutletShutterCom2.tyBitmapMc.uiValueIdx	:= tyP0921InletNOutletShutter.tyOutletShutterCom2.tyBitmapMc.uiValueIdx + 701;
			END_IF
		ELSIF p_tyNtParamCurr.bProjLifterMagPlatform AND p_tyNtParamCurr.bUIConvDirRL = FALSE AND p_tyNtParamCurr.bProjMagConvLane1Prep THEN
			IF 	tyP0921InletNOutletShutter.tyOutletShutterCom2.tyBitmapMc.uiValueIdx < 100 THEN
				tyP0921InletNOutletShutter.tyOutletShutterCom2.tyBitmapMc.uiValueIdx	:= tyP0921InletNOutletShutter.tyOutletShutterCom2.tyBitmapMc.uiValueIdx + 901;
			END_IF
		ELSIF p_tyNtParamCurr.bProjLifterMagPlatform THEN
				IF 	tyP0921InletNOutletShutter.tyOutletShutterCom2.tyBitmapMc.uiValueIdx < 100 THEN
					tyP0921InletNOutletShutter.tyOutletShutterCom2.tyBitmapMc.uiValueIdx	:= tyP0921InletNOutletShutter.tyOutletShutterCom2.tyBitmapMc.uiValueIdx + 601;
				END_IF
		ELSIF p_tyNtParamCurr.bProjMagAWPrep = FALSE THEN
			tyP0921InletNOutletShutter.tyOutletShutterCom2.tyBitmapMc.uiValueIdx	:= tyP0921InletNOutletShutter.tyOutletShutterCom2.tyBitmapMc.uiValueIdx + 4;
		ELSIF p_tyNtParamCurr.bProjMagAWPrep THEN
			tyP0921InletNOutletShutter.tyOutletShutterCom2.tyBitmapMc.uiValueIdx	:= tyP0921InletNOutletShutter.tyOutletShutterCom2.tyBitmapMc.uiValueIdx + 335;
		END_IF
	END_IF

END_ACTION
```

#### Act_OptP0921OutletShutterFB2.st
```iecst
ACTION Act_OptP0921OutletShutterFB2:

	IF tyP0921InletNOutletShutter.tyOutletShutterCom2.tyBtnSwitch.bValue = FALSE THEN
		// FB Control
		IF tyP0921InletNOutletShutter.tyOutletShutterFB2.tyBtnOpen.bRtCompl = TRUE THEN
			tyP0921InletNOutletShutter.tyOutletShutterFB2.tyBtnOpen.bRtCompl	:= FALSE;

			tyP0921InletNOutletShutter.tyOutletShutterFB2.tyBtnOpen.bValue	:= TRUE;
			tyP0921InletNOutletShutter.tyOutletShutterFB2.tyBtnClose.bValue	:= FALSE;

		ELSIF tyP0921InletNOutletShutter.tyOutletShutterFB2.tyBtnClose.bRtCompl = TRUE THEN
			tyP0921InletNOutletShutter.tyOutletShutterFB2.tyBtnClose.bRtCompl	:= FALSE;

			tyP0921InletNOutletShutter.tyOutletShutterFB2.tyBtnClose.bValue	:= TRUE;
			tyP0921InletNOutletShutter.tyOutletShutterFB2.tyBtnOpen.bValue	:= FALSE;
		END_IF

		IF tyP0921InletNOutletShutter.tyOutletShutterFB2.tyBtnOpen.bValue = TRUE THEN
			eOutShutterAct2	:= PneuActRet;

			IF p_eOutShutterStat2 = PneuActRet AND p_eOutShutterStatus2 = Done THEN
				eOutShutterAct2	:= PneuActIdle;

				tyP0921InletNOutletShutter.tyOutletShutterFB2.tyBtnOpen.bValue	:= FALSE;
			ELSIF p_eOutShutterStatus2 = Error THEN
				tyP0921InletNOutletShutter.tyOutletShutterFB2.tyBtnOpen.bValue	:= FALSE;
			END_IF

		ELSIF tyP0921InletNOutletShutter.tyOutletShutterFB2.tyBtnClose.bValue = TRUE THEN
			eOutShutterAct2		:= PneuActExt;

			IF p_eOutShutterStat2 = PneuActExt AND p_eOutShutterStatus2 = Done THEN

				eOutShutterAct2	:= PneuActIdle;

				tyP0921InletNOutletShutter.tyOutletShutterFB2.tyBtnClose.bValue := FALSE;
			ELSIF p_eOutShutterStatus2 = Error THEN
				tyP0921InletNOutletShutter.tyOutletShutterFB2.tyBtnClose.bValue := FALSE;
			END_IF

		END_IF

		//UpdateStatus
		tyP0921InletNOutletShutter.tyOutletShutterDC2.tyBtnClose.bRtCompl		:= FALSE;
		tyP0921InletNOutletShutter.tyOutletShutterDC2.tyBtnOpen.bRtCompl		:= FALSE;
		tyP0921InletNOutletShutter.tyOutletShutterDC2.tyBtnClose.bValue			:= p_bOutShutterExtCtrl2;
		tyP0921InletNOutletShutter.tyOutletShutterDC2.tyBtnOpen.bValue			:= p_bOutShutterRetCtrl2;

	END_IF

END_ACTION
```

#### Act_OptP0921OutletShutterFBStat2.st
```iecst
ACTION Act_OptP0921OutletShutterFBStat2:

	tyP0921InletNOutletShutter.tyOutletShutterFB2.tyStringStat.sValue	:= p_sOutShutterStatTxt2;

END_ACTION
```

#### Act_OptP0921OutletShutterDC2.st
```iecst
ACTION Act_OptP0921OutletShutterDC2:

	// Direct Control
	IF tyP0921InletNOutletShutter.tyOutletShutterCom2.tyBtnSwitch.bValue = TRUE THEN
		IF p_bOutShutterTwoCtrlOut2 = FALSE THEN
			IF tyP0921InletNOutletShutter.tyOutletShutterDC2.tyBtnOpen.bRtCompl = TRUE THEN
				tyP0921InletNOutletShutter.tyOutletShutterDC2.tyBtnOpen.bValue	:= TRUE;
				tyP0921InletNOutletShutter.tyOutletShutterDC2.tyBtnClose.bValue	:= FALSE;

				eOutShutterAct2	:= PneuActSetRet;

				IF p_eOutShutterStat2 = PneuActSetRet AND p_eOutShutterStatus2 = Done THEN
					eOutShutterAct2	:= PneuActIdle;

					tyP0921InletNOutletShutter.tyOutletShutterDC2.tyBtnOpen.bRtCompl	:= FALSE;
				END_IF

			ELSIF tyP0921InletNOutletShutter.tyOutletShutterDC2.tyBtnClose.bRtCompl = TRUE THEN
				tyP0921InletNOutletShutter.tyOutletShutterDC2.tyBtnClose.bValue	:= TRUE;
				tyP0921InletNOutletShutter.tyOutletShutterDC2.tyBtnOpen.bValue	:= FALSE;

				eOutShutterAct2	:= PneuActSetExt;

				IF p_eOutShutterStat2 = PneuActSetExt AND p_eOutShutterStatus2 = Done THEN
					eOutShutterAct2	:= PneuActIdle;

					tyP0921InletNOutletShutter.tyOutletShutterDC2.tyBtnClose.bRtCompl	:= FALSE;
				END_IF
			END_IF

		ELSE
			IF (tyP0921InletNOutletShutter.tyOutletShutterDC2.tyBtnOpen.bRtCompl = TRUE) OR (tyP0921InletNOutletShutter.tyOutletShutterDC2.tyBtnClose.bRtCompl = TRUE) THEN
				IF (tyP0921InletNOutletShutter.tyOutletShutterDC2.tyBtnOpen.bValue = TRUE) AND (tyP0921InletNOutletShutter.tyOutletShutterDC2.tyBtnClose.bValue = TRUE) THEN
					eOutShutterAct2	:= PneuActSetAll;

					IF p_eOutShutterStat2 = PneuActSetAll AND p_eOutShutterStatus2 = Done THEN
						eOutShutterAct2	:= PneuActIdle;

						tyP0921InletNOutletShutter.tyOutletShutterDC2.tyBtnOpen.bRtCompl		:= FALSE;
						tyP0921InletNOutletShutter.tyOutletShutterDC2.tyBtnClose.bRtCompl	:= FALSE;
					END_IF

				ELSIF (tyP0921InletNOutletShutter.tyOutletShutterDC2.tyBtnOpen.bValue = TRUE) AND (tyP0921InletNOutletShutter.tyOutletShutterDC2.tyBtnClose.bValue = FALSE) THEN
					eOutShutterAct2	:= PneuActSetRet;

					IF p_eOutShutterStat2 = PneuActSetRet AND p_eOutShutterStatus2 = Done THEN
						eOutShutterAct2	:= PneuActIdle;

						tyP0921InletNOutletShutter.tyOutletShutterDC2.tyBtnOpen.bRtCompl		:= FALSE;
						tyP0921InletNOutletShutter.tyOutletShutterDC2.tyBtnClose.bRtCompl	:= FALSE;
					END_IF

				ELSIF (tyP0921InletNOutletShutter.tyOutletShutterDC2.tyBtnOpen.bValue = FALSE) AND (tyP0921InletNOutletShutter.tyOutletShutterDC2.tyBtnClose.bValue = TRUE) THEN
					eOutShutterAct2	:= PneuActSetExt;

					IF p_eOutShutterStat2 = PneuActSetExt AND p_eOutShutterStatus2 = Done THEN
						eOutShutterAct2	:= PneuActIdle;

						tyP0921InletNOutletShutter.tyOutletShutterDC2.tyBtnOpen.bRtCompl		:= FALSE;
						tyP0921InletNOutletShutter.tyOutletShutterDC2.tyBtnClose.bRtCompl	:= FALSE;
					END_IF

				ELSE
					eOutShutterAct2	:= PneuActRstAll;

					IF p_eOutShutterStat2 = PneuActRstAll AND p_eOutShutterStatus2 = Done THEN
						eOutShutterAct2	:= PneuActIdle;

						tyP0921InletNOutletShutter.tyOutletShutterDC2.tyBtnOpen.bRtCompl		:= FALSE;
						tyP0921InletNOutletShutter.tyOutletShutterDC2.tyBtnClose.bRtCompl	:= FALSE;
					END_IF

				END_IF
			END_IF
		END_IF

		tyP0921InletNOutletShutter.tyOutletShutterFB2.tyBtnOpen.bRtCompl	:= FALSE;
		tyP0921InletNOutletShutter.tyOutletShutterFB2.tyBtnOpen.bValue	:= FALSE;
		tyP0921InletNOutletShutter.tyOutletShutterFB2.tyBtnClose.bRtCompl:= FALSE;
		tyP0921InletNOutletShutter.tyOutletShutterFB2.tyBtnClose.bValue	:= FALSE;

	END_IF

END_ACTION
```

#### Act_EntP0922Disp.st
```iecst
ACTION Act_EntP0922Disp:

	//Access Address
	p_tyC0003DualMask ACCESS ADR(tyP0922Stopper.tyDualMaskHide);

	p_tyC0004Navi ACCESS ADR(tyP0921InletNOutletShutter.tyNaviBack);

	p_tyC0005Main ACCESS ADR(tyCommon.tyMain);

	p_tyC0007Notif ACCESS ADR(tyCommon.tyNotif);

	p_tyC0008MsgBox ACCESS ADR(tyP0921InletNOutletShutter.tyMsgBoxHide);

	p_tyC0009Info ACCESS ADR(tyCommon.tyInfo);

	IF (p_tyNtParamCurr.bProjStopperAPrep OR p_tyNtParamCurr.bProjStopperBPrep ) THEN
		p_tyP0922StopperACom ACCESS ADR(tyP0922Stopper.tyStopperACom);
		p_tyP0922StopperADC ACCESS ADR(tyP0922Stopper.tyStopperADC);
		p_tyP0922StopperAFB ACCESS ADR(tyP0922Stopper.tyStopperAFB);
		p_tyP0922StopperADis ACCESS ADR(tyP0922Stopper.tyStopperADis);

		p_tyP0922StopperBCom ACCESS ADR(tyP0922Stopper.tyStopperBCom);
		p_tyP0922StopperBDC ACCESS ADR(tyP0922Stopper.tyStopperBDC);
		p_tyP0922StopperBFB ACCESS ADR(tyP0922Stopper.tyStopperBFB);
		p_tyP0922StopperBDis ACCESS ADR(tyP0922Stopper.tyStopperBDis);

	ELSIF p_tyNtParamCurr.bProjInletStopperPrep THEN

		p_tyP0922StopperACom ACCESS ADR(tyP0922Stopper.tyInStopperCom);
		p_tyP0922StopperADC ACCESS ADR(tyP0922Stopper.tyInStopperDC);
		p_tyP0922StopperAFB ACCESS ADR(tyP0922Stopper.tyInStopperFB);
		p_tyP0922StopperADis ACCESS ADR(tyP0922Stopper.tyInStopperDis);

		p_tyP0922StopperBCom ACCESS ADR(tyP0922Stopper.tyStopperBCom); //can be replaced by other if needed
		p_tyP0922StopperBDC ACCESS ADR(tyP0922Stopper.tyStopperBDC); //can be replaced by other if needed
		p_tyP0922StopperBFB ACCESS ADR(tyP0922Stopper.tyStopperBFB); //can be replaced by other if needed
		p_tyP0922StopperBDis ACCESS ADR(tyP0922Stopper.tyStopperBDis); //can be replaced by other if needed
	END_IF
	//Display
	tyP0922Stopper.tyStopperADis.tyLyr.uiRtStat.0	:= NOT(p_tyNtParamCurr.bProjStopperAPrep AND p_tyMcParamCurr.bStopperADis);

	tyP0922Stopper.tyStopperBDis.tyLyr.uiRtStat.0	:= NOT(p_tyNtParamCurr.bProjStopperBPrep AND p_tyMcParamCurr.bStopperBDis);

	tyP0922Stopper.tyInStopperDis.tyLyr.uiRtStat.0   := NOT(p_tyNtParamCurr.bProjInletStopperPrep AND p_tyMcParamCurr.bInStopperDis);
END_ACTION
```

#### Act_OptP0922Navi.st
```iecst
ACTION Act_OptP0922Navi:

	IF tyP0922Stopper.tyNaviBack.tyBtnBack.bRtCompl = TRUE THEN
		eChgPage		:= UIP0920MtrNPneuCtrl;

		tyP0922Stopper.tyNaviBack.tyBtnBack.bRtCompl 	:= FALSE;
		tyP0922Stopper.tyNaviBack.tyBtnBack.bValue		:= FALSE;
	END_IF

END_ACTION
```

#### Act_OptP0922DualMask.st
```iecst
ACTION Act_OptP0922DualMask:

	IF eCurrPage = UIP0922Stopper THEN

		IF p_tyDI.bEStopSig = FALSE THEN
			p_tyC0003DualMask ACCESS ADR(tyP0922Stopper.tyDualMaskEStop);

			tyP0922Stopper.tyDualMaskEStop.tyBtnLeftMask.uiMaskRtStat.0	:= NOT p_tyNtParamCurr.bProjStopperAPrep;
			tyP0922Stopper.tyDualMaskEStop.tyBtnRgtMask.uiMaskRtStat.0	:= NOT p_tyNtParamCurr.bProjStopperBPrep;

		ELSIF p_tyDI.bCoverSWSig = FALSE THEN
			p_tyC0003DualMask ACCESS ADR(tyP0922Stopper.tyDualMaskCWSig);

			tyP0922Stopper.tyDualMaskCWSig.tyBtnLeftMask.uiMaskRtStat.0	:= NOT p_tyNtParamCurr.bProjStopperAPrep;
			tyP0922Stopper.tyDualMaskCWSig.tyBtnRgtMask.uiMaskRtStat.0	:= NOT p_tyNtParamCurr.bProjStopperBPrep;

		ELSIF p_tyDI.bSafetyRlySig = FALSE THEN
			p_tyC0003DualMask ACCESS ADR(tyP0922Stopper.tyDualMaskSafetyRly);

			tyP0922Stopper.tyDualMaskSafetyRly.tyBtnLeftMask.uiMaskRtStat.0	:= NOT p_tyNtParamCurr.bProjStopperAPrep;
			tyP0922Stopper.tyDualMaskSafetyRly.tyBtnRgtMask.uiMaskRtStat.0	:= NOT p_tyNtParamCurr.bProjStopperBPrep;

		ELSE
			p_tyC0003DualMask ACCESS ADR(tyP0922Stopper.tyDualMaskHide);

		END_IF

	END_IF

END_ACTION
```

#### Act_OptP0922StopperAChgLyr.st
```iecst
ACTION Act_OptP0922StopperAChgLyr:
	IF p_tyNtParamCurr.bProjStopperAPrep   THEN
		IF tyP0922Stopper.tyStopperACom.tyBtnSwitch.bValue = TRUE THEN
			fUIInRtStatOff(ADR(tyP0922Stopper.tyStopperADC.tyLyr.uiRtStat));
			fUIInRtStatHide(ADR(tyP0922Stopper.tyStopperAFB.tyLyr.uiRtStat));
		ELSE
			fUIInRtStatHide(ADR(tyP0922Stopper.tyStopperADC.tyLyr.uiRtStat));
			fUIInRtStatOff(ADR(tyP0922Stopper.tyStopperAFB.tyLyr.uiRtStat));
		END_IF
	END_IF

END_ACTION
```

#### Act_OptP0922StopperASen.st
```iecst
ACTION Act_OptP0922StopperASen:

	//tyP0921InletNOutletShutter.tyInletShutterCom.tyBtnOpenRS.bValue	:= p_tyDI.bInShutterOpenRS;
	//tyP0921InletNOutletShutter.tyInletShutterCom.tyBtnCloseRS.bValue	:= p_tyDI.bInShutterCloseRS;

END_ACTION
```

#### Act_OptP0922StopperAFB.st
```iecst
ACTION Act_OptP0922StopperAFB:

	IF tyP0922Stopper.tyStopperACom.tyBtnSwitch.bValue = FALSE THEN

		// FB Control
		IF tyP0922Stopper.tyStopperAFB.tyBtnUnblk.bRtCompl = TRUE THEN
			tyP0922Stopper.tyStopperAFB.tyBtnUnblk.bRtCompl	:= FALSE;

			tyP0922Stopper.tyStopperAFB.tyBtnUnblk.bValue	:= TRUE;
			tyP0922Stopper.tyStopperAFB.tyBtnBlk.bValue		:= FALSE;

		ELSIF tyP0922Stopper.tyStopperAFB.tyBtnBlk.bRtCompl = TRUE THEN
			tyP0922Stopper.tyStopperAFB.tyBtnBlk.bRtCompl	:= FALSE;

			tyP0922Stopper.tyStopperAFB.tyBtnBlk.bValue		:= TRUE;
			tyP0922Stopper.tyStopperAFB.tyBtnUnblk.bValue	:= FALSE;
		END_IF

		IF tyP0922Stopper.tyStopperAFB.tyBtnUnblk.bValue = TRUE THEN

			eStopperAAct	:= PneuActRet;

			IF p_eStopperAStat = PneuActRet AND p_eStopperAStatus = Done THEN
				eStopperAAct	:= PneuActIdle;

				tyP0922Stopper.tyStopperAFB.tyBtnUnblk.bValue	:= FALSE;

			ELSIF p_eStopperAStatus = Error THEN
				tyP0922Stopper.tyStopperAFB.tyBtnUnblk.bValue	:= FALSE;
			END_IF

		ELSIF tyP0922Stopper.tyStopperAFB.tyBtnBlk.bValue = TRUE THEN
			eStopperAAct	:= PneuActExt;

			IF p_eStopperAStat = PneuActExt AND p_eStopperAStatus = Done THEN
				eStopperAAct	:= PneuActIdle;

				tyP0922Stopper.tyStopperAFB.tyBtnBlk.bValue := FALSE;
			ELSIF p_eStopperAStatus = Error THEN
				tyP0922Stopper.tyStopperAFB.tyBtnBlk.bValue := FALSE;
			END_IF
		END_IF
		//Update Status

		tyP0922Stopper.tyStopperADC.tyBtnUnblk.bRtCompl		:= FALSE;
		tyP0922Stopper.tyStopperADC.tyBtnBlk.bRtCompl		:= FALSE;
		tyP0922Stopper.tyStopperADC.tyBtnUnblk.bValue		:= p_bStopperARetCtrl;
		tyP0922Stopper.tyStopperADC.tyBtnBlk.bValue			:= NOT p_bStopperARetCtrl;

	END_IF

END_ACTION
```

#### Act_OptP0922StopperAFBStat.st
```iecst
ACTION Act_OptP0922StopperAFBStat:

	tyP0922Stopper.tyStopperAFB.tyStringStat.sValue	:= p_sStopperAStatTxt;

END_ACTION
```

#### Act_OptP0922StopperADC.st
```iecst
ACTION Act_OptP0922StopperADC:

	IF tyP0922Stopper.tyStopperACom.tyBtnSwitch.bValue = TRUE THEN
		// Direct Control
		IF p_bStopperATwoCtrlOut = FALSE THEN
			IF tyP0922Stopper.tyStopperADC.tyBtnUnblk.bRtCompl = TRUE THEN
				tyP0922Stopper.tyStopperADC.tyBtnUnblk.bValue	:= TRUE;
				tyP0922Stopper.tyStopperADC.tyBtnBlk.bValue		:= FALSE;

				eStopperAAct	:= PneuActSetRet;

				IF p_eStopperAStat = PneuActSetRet AND p_eStopperAStatus = Done THEN
					eStopperAAct	:= PneuActIdle;

					tyP0922Stopper.tyStopperADC.tyBtnUnblk.bRtCompl	:= FALSE;
				END_IF

			ELSIF tyP0922Stopper.tyStopperADC.tyBtnBlk.bRtCompl = TRUE THEN
				tyP0922Stopper.tyStopperADC.tyBtnBlk.bValue		:= TRUE;
				tyP0922Stopper.tyStopperADC.tyBtnUnblk.bValue	:= FALSE;

				eStopperAAct	:= PneuActSetExt;

				IF p_eStopperAStat = PneuActSetExt AND p_eStopperAStatus = Done THEN
					eStopperAAct	:= PneuActIdle;

					tyP0922Stopper.tyStopperADC.tyBtnBlk.bRtCompl	:= FALSE;
				END_IF
			END_IF

		ELSE
			IF (tyP0922Stopper.tyStopperADC.tyBtnUnblk.bRtCompl = TRUE) OR (tyP0922Stopper.tyStopperADC.tyBtnBlk.bRtCompl = TRUE) THEN
				IF (tyP0922Stopper.tyStopperADC.tyBtnUnblk.bValue = TRUE) AND (tyP0922Stopper.tyStopperADC.tyBtnBlk.bValue = TRUE) THEN

					eStopperAAct	:= PneuActSetAll;

					IF p_eStopperAStat = PneuActSetAll AND p_eStopperAStatus = Done THEN
						eStopperAAct	:= PneuActIdle;

						tyP0922Stopper.tyStopperADC.tyBtnUnblk.bRtCompl	:= FALSE;
						tyP0922Stopper.tyStopperADC.tyBtnBlk.bRtCompl	:= FALSE;
					END_IF

				ELSIF (tyP0922Stopper.tyStopperADC.tyBtnUnblk.bValue = TRUE) AND (tyP0922Stopper.tyStopperADC.tyBtnBlk.bValue = FALSE) THEN

					eStopperAAct	:= PneuActSetRet;

					IF p_eStopperAStat = PneuActSetRet AND p_eStopperAStatus = Done THEN

						eStopperAAct	:= PneuActIdle;

						tyP0922Stopper.tyStopperADC.tyBtnUnblk.bRtCompl	:= FALSE;
						tyP0922Stopper.tyStopperADC.tyBtnBlk.bRtCompl	:= FALSE;
					END_IF

				ELSIF (tyP0922Stopper.tyStopperADC.tyBtnUnblk.bValue = FALSE) AND (tyP0922Stopper.tyStopperADC.tyBtnBlk.bValue = TRUE) THEN

					eStopperAAct	:= PneuActSetExt;

					IF p_eStopperAStat = PneuActSetExt AND p_eStopperAStatus = Done THEN
						eStopperAAct	:= PneuActIdle;

						tyP0922Stopper.tyStopperADC.tyBtnUnblk.bRtCompl	:= FALSE;
						tyP0922Stopper.tyStopperADC.tyBtnBlk.bRtCompl	:= FALSE;
					END_IF

				ELSE
					eStopperAAct	:= PneuActRstAll;

					IF p_eStopperAStat = PneuActRstAll AND p_eStopperAStatus = Done THEN
						eStopperAAct	:= PneuActIdle;

						tyP0922Stopper.tyStopperADC.tyBtnUnblk.bRtCompl	:= FALSE;
						tyP0922Stopper.tyStopperADC.tyBtnBlk.bRtCompl	:= FALSE;
					END_IF

				END_IF
			END_IF
		END_IF

		//Update Status
		tyP0922Stopper.tyStopperAFB.tyBtnUnblk.bValue		:= FALSE;
		tyP0922Stopper.tyStopperAFB.tyBtnBlk.bValue			:= FALSE;
		tyP0922Stopper.tyStopperAFB.tyBtnUnblk.bRtCompl		:= FALSE;
		tyP0922Stopper.tyStopperAFB.tyBtnBlk.bRtCompl		:= FALSE;

	END_IF

END_ACTION
```

#### Act_OptP0922StopperBChgLyr.st
```iecst
ACTION Act_OptP0922StopperBChgLyr:
	IF p_tyNtParamCurr.bProjStopperBPrep THEN
		IF tyP0922Stopper.tyStopperBCom.tyBtnSwitch.bValue = TRUE THEN
			fUIInRtStatOff(ADR(tyP0922Stopper.tyStopperBDC.tyLyr.uiRtStat));
			fUIInRtStatHide(ADR(tyP0922Stopper.tyStopperBFB.tyLyr.uiRtStat));
		ELSE
			fUIInRtStatHide(ADR(tyP0922Stopper.tyStopperBDC.tyLyr.uiRtStat));
			fUIInRtStatOff(ADR(tyP0922Stopper.tyStopperBFB.tyLyr.uiRtStat));
		END_IF
	END_IF

END_ACTION
```

#### Act_OptP0922StopperBSen.st
```iecst
ACTION Act_OptP0922StopperBSen:

	//tyP0921InletNOutletShutter.tyInletShutterCom.tyBtnOpenRS.bValue		:= p_tyDI.bInShutterOpenRS;
	//tyP0921InletNOutletShutter.tyInletShutterCom.tyBtnCloseRS.bValue	:= p_tyDI.bInShutterCloseRS;

END_ACTION
```

#### Act_OptP0922StopperBFB.st
```iecst
ACTION Act_OptP0922StopperBFB:

	IF tyP0922Stopper.tyStopperBCom.tyBtnSwitch.bValue = FALSE THEN

		// FB Control
		IF tyP0922Stopper.tyStopperBFB.tyBtnUnblk.bRtCompl = TRUE THEN
			tyP0922Stopper.tyStopperBFB.tyBtnUnblk.bRtCompl	:= FALSE;

			tyP0922Stopper.tyStopperBFB.tyBtnUnblk.bValue	:= TRUE;
			tyP0922Stopper.tyStopperBFB.tyBtnBlk.bValue		:= FALSE;

		ELSIF tyP0922Stopper.tyStopperBFB.tyBtnBlk.bRtCompl = TRUE THEN
			tyP0922Stopper.tyStopperBFB.tyBtnBlk.bRtCompl	:= FALSE;

			tyP0922Stopper.tyStopperBFB.tyBtnBlk.bValue		:= TRUE;
			tyP0922Stopper.tyStopperBFB.tyBtnUnblk.bValue	:= FALSE;
		END_IF

		IF tyP0922Stopper.tyStopperBFB.tyBtnUnblk.bValue = TRUE THEN

			eStopperBAct	:= PneuActRet;

			IF p_eStopperBStat = PneuActRet AND p_eStopperBStatus = Done THEN
				eStopperBAct	:= PneuActIdle;

				tyP0922Stopper.tyStopperBFB.tyBtnUnblk.bValue	:= FALSE;

			ELSIF p_eStopperBStatus = Error THEN
				tyP0922Stopper.tyStopperBFB.tyBtnUnblk.bValue	:= FALSE;
			END_IF

		ELSIF tyP0922Stopper.tyStopperBFB.tyBtnBlk.bValue = TRUE THEN
			eStopperBAct	:= PneuActExt;

			IF p_eStopperBStat = PneuActExt AND p_eStopperBStatus = Done THEN
				eStopperBAct	:= PneuActIdle;

				tyP0922Stopper.tyStopperBFB.tyBtnBlk.bValue := FALSE;
			ELSIF p_eStopperBStatus = Error THEN
				tyP0922Stopper.tyStopperBFB.tyBtnBlk.bValue := FALSE;
			END_IF
		END_IF

		//Update Status
		tyP0922Stopper.tyStopperBDC.tyBtnUnblk.bRtCompl		:= FALSE;
		tyP0922Stopper.tyStopperBDC.tyBtnBlk.bRtCompl		:= FALSE;
		tyP0922Stopper.tyStopperBDC.tyBtnUnblk.bValue		:= p_bStopperBRetCtrl;
		tyP0922Stopper.tyStopperBDC.tyBtnBlk.bValue			:= NOT p_bStopperBRetCtrl;

	END_IF

END_ACTION
```

#### Act_OptP0922StopperBFBStat.st
```iecst
ACTION Act_OptP0922StopperBFBStat:

	tyP0922Stopper.tyStopperBFB.tyStringStat.sValue	:= p_sStopperBStatTxt;

END_ACTION
```

#### Act_OptP0922StopperBDC.st
```iecst
ACTION Act_OptP0922StopperBDC:

	IF tyP0922Stopper.tyStopperBCom.tyBtnSwitch.bValue = TRUE THEN
		// Direct Control
		IF p_bStopperBTwoCtrlOut = FALSE THEN
			IF tyP0922Stopper.tyStopperBDC.tyBtnUnblk.bRtCompl = TRUE THEN
				tyP0922Stopper.tyStopperBDC.tyBtnUnblk.bValue	:= TRUE;
				tyP0922Stopper.tyStopperBDC.tyBtnBlk.bValue		:= FALSE;

				eStopperBAct	:= PneuActSetRet;

				IF p_eStopperBStat = PneuActSetRet AND p_eStopperBStatus = Done THEN
					eStopperBAct	:= PneuActIdle;

					tyP0922Stopper.tyStopperBDC.tyBtnUnblk.bRtCompl	:= FALSE;
				END_IF

			ELSIF tyP0922Stopper.tyStopperBDC.tyBtnBlk.bRtCompl = TRUE THEN
				tyP0922Stopper.tyStopperBDC.tyBtnBlk.bValue		:= TRUE;
				tyP0922Stopper.tyStopperBDC.tyBtnUnblk.bValue	:= FALSE;

				eStopperBAct	:= PneuActSetExt;

				IF p_eStopperBStat = PneuActSetExt AND p_eStopperBStatus = Done THEN
					eStopperBAct	:= PneuActIdle;

					tyP0922Stopper.tyStopperBDC.tyBtnBlk.bRtCompl	:= FALSE;
				END_IF
			END_IF

		ELSE
			IF (tyP0922Stopper.tyStopperBDC.tyBtnUnblk.bRtCompl = TRUE) OR (tyP0922Stopper.tyStopperBDC.tyBtnBlk.bRtCompl = TRUE) THEN
				IF (tyP0922Stopper.tyStopperBDC.tyBtnUnblk.bValue = TRUE) AND (tyP0922Stopper.tyStopperBDC.tyBtnBlk.bValue = TRUE) THEN

					eStopperBAct	:= PneuActSetAll;

					IF p_eStopperBStat = PneuActSetAll AND p_eStopperBStatus = Done THEN
						eStopperBAct	:= PneuActIdle;

						tyP0922Stopper.tyStopperBDC.tyBtnUnblk.bRtCompl	:= FALSE;
						tyP0922Stopper.tyStopperBDC.tyBtnBlk.bRtCompl	:= FALSE;
					END_IF

				ELSIF (tyP0922Stopper.tyStopperBDC.tyBtnUnblk.bValue = TRUE) AND (tyP0922Stopper.tyStopperBDC.tyBtnBlk.bValue = FALSE) THEN

					eStopperBAct	:= PneuActSetRet;

					IF p_eStopperBStat = PneuActSetRet AND p_eStopperBStatus = Done THEN

						eStopperBAct	:= PneuActIdle;

						tyP0922Stopper.tyStopperBDC.tyBtnUnblk.bRtCompl	:= FALSE;
						tyP0922Stopper.tyStopperBDC.tyBtnBlk.bRtCompl	:= FALSE;
					END_IF

				ELSIF (tyP0922Stopper.tyStopperBDC.tyBtnUnblk.bValue = FALSE) AND (tyP0922Stopper.tyStopperBDC.tyBtnBlk.bValue = TRUE) THEN

					eStopperBAct	:= PneuActSetExt;

					IF p_eStopperBStat = PneuActSetExt AND p_eStopperBStatus = Done THEN
						eStopperBAct	:= PneuActIdle;

						tyP0922Stopper.tyStopperBDC.tyBtnUnblk.bRtCompl	:= FALSE;
						tyP0922Stopper.tyStopperBDC.tyBtnBlk.bRtCompl	:= FALSE;
					END_IF

				ELSE
					eStopperBAct	:= PneuActRstAll;

					IF p_eStopperBStat = PneuActRstAll AND p_eStopperBStatus = Done THEN
						eStopperBAct	:= PneuActIdle;

						tyP0922Stopper.tyStopperBDC.tyBtnUnblk.bRtCompl	:= FALSE;
						tyP0922Stopper.tyStopperBDC.tyBtnBlk.bRtCompl	:= FALSE;
					END_IF

				END_IF
			END_IF

			//Update Status
			tyP0922Stopper.tyStopperBFB.tyBtnUnblk.bRtCompl		:= FALSE;
			tyP0922Stopper.tyStopperBFB.tyBtnBlk.bRtCompl		:= FALSE;
			tyP0922Stopper.tyStopperBFB.tyBtnUnblk.bValue		:= FALSE;
			tyP0922Stopper.tyStopperBFB.tyBtnBlk.bValue			:= FALSE;

		END_IF
	END_IF

END_ACTION
```

#### Act_OptP0922InStopperChgLyr.st
```iecst
ACTION Act_OptP0922InStopperChgLyr:
	IF p_tyNtParamCurr.bProjInletStopperPrep THEN
		IF tyP0922Stopper.tyInStopperCom.tyBtnSwitch.bValue = TRUE THEN
			fUIInRtStatOff(ADR(tyP0922Stopper.tyInStopperDC.tyLyr.uiRtStat));
			fUIInRtStatHide(ADR(tyP0922Stopper.tyInStopperFB.tyLyr.uiRtStat));
		ELSE
			fUIInRtStatHide(ADR(tyP0922Stopper.tyInStopperDC.tyLyr.uiRtStat));
			fUIInRtStatOff(ADR(tyP0922Stopper.tyInStopperFB.tyLyr.uiRtStat));
		END_IF
	END_IF

END_ACTION
```

#### Act_OptP0922InStopperSen.st
```iecst
ACTION Act_OptP0922InStopperSen:

	//tyP0921InletNOutletShutter.tyInletShutterCom.tyBtnOpenRS.bValue	:= p_tyDI.bInShutterOpenRS;
	//tyP0921InletNOutletShutter.tyInletShutterCom.tyBtnCloseRS.bValue	:= p_tyDI.bInShutterCloseRS;

	IF p_InletStopperRetCtrl = TRUE THEN
		tyP0922Stopper.tyInStopperCom.tyBitmapMc.uiValueIdx := 0;
	ELSE
		tyP0922Stopper.tyInStopperCom.tyBitmapMc.uiValueIdx := 1;
	END_IF

END_ACTION
```

#### Act_OptP0922InStopperFB.st
```iecst
ACTION Act_OptP0922InStopperFB:

	IF tyP0922Stopper.tyInStopperCom.tyBtnSwitch.bValue = FALSE THEN

		// FB Control
		IF tyP0922Stopper.tyInStopperFB.tyBtnUnblk.bRtCompl = TRUE THEN
			tyP0922Stopper.tyInStopperFB.tyBtnUnblk.bRtCompl	:= FALSE;

			tyP0922Stopper.tyInStopperFB.tyBtnUnblk.bValue	:= TRUE;
			tyP0922Stopper.tyInStopperFB.tyBtnBlk.bValue		:= FALSE;

		ELSIF tyP0922Stopper.tyInStopperFB.tyBtnBlk.bRtCompl = TRUE THEN
			tyP0922Stopper.tyInStopperFB.tyBtnBlk.bRtCompl	:= FALSE;

			tyP0922Stopper.tyInStopperFB.tyBtnBlk.bValue		:= TRUE;
			tyP0922Stopper.tyInStopperFB.tyBtnUnblk.bValue	:= FALSE;
		END_IF

		IF tyP0922Stopper.tyInStopperFB.tyBtnUnblk.bValue = TRUE THEN

			eInStopperAct	:= PneuActRet;

			IF p_eInStopperStat = PneuActRet AND p_eInStopperStatus = Done THEN
				eInStopperAct	:= PneuActIdle;

				tyP0922Stopper.tyInStopperFB.tyBtnUnblk.bValue	:= FALSE;

			ELSIF p_eInStopperStatus = Error THEN
				tyP0922Stopper.tyInStopperFB.tyBtnUnblk.bValue	:= FALSE;
			END_IF

		ELSIF tyP0922Stopper.tyInStopperFB.tyBtnBlk.bValue = TRUE THEN
			eInStopperAct	:= PneuActExt;

			IF p_eInStopperStat = PneuActExt AND p_eInStopperStatus = Done THEN
				eInStopperAct	:= PneuActIdle;

				tyP0922Stopper.tyInStopperFB.tyBtnBlk.bValue := FALSE;
			ELSIF p_eInStopperStatus = Error THEN
				tyP0922Stopper.tyInStopperFB.tyBtnBlk.bValue := FALSE;
			END_IF
		END_IF
		//Update Status

		tyP0922Stopper.tyInStopperDC.tyBtnUnblk.bRtCompl		:= FALSE;
		tyP0922Stopper.tyInStopperDC.tyBtnBlk.bRtCompl		:= FALSE;
		tyP0922Stopper.tyInStopperDC.tyBtnUnblk.bValue		:= p_bInStopperRetCtrl;
		tyP0922Stopper.tyInStopperDC.tyBtnBlk.bValue			:= NOT p_bInStopperRetCtrl;

	END_IF

END_ACTION
```

#### Act_OptP0922InStopperFBStat.st
```iecst
ACTION Act_OptP0922InStopperFBStat:

	tyP0922Stopper.tyInStopperFB.tyStringStat.sValue	:= p_sInStopperStatTxt;

END_ACTION
```

#### Act_OptP0922InStopperDC.st
```iecst
ACTION Act_OptP0922InStopperDC:

	IF tyP0922Stopper.tyInStopperCom.tyBtnSwitch.bValue = TRUE THEN
		// Direct Control
		IF p_bInStopperTwoCtrlOut = FALSE THEN
			IF tyP0922Stopper.tyInStopperDC.tyBtnUnblk.bRtCompl = TRUE THEN
				tyP0922Stopper.tyInStopperDC.tyBtnUnblk.bValue	:= TRUE;
				tyP0922Stopper.tyInStopperDC.tyBtnBlk.bValue		:= FALSE;

				eInStopperAct	:= PneuActSetRet;

				IF p_eInStopperStat = PneuActSetRet AND p_eInStopperStatus = Done THEN
					eInStopperAct	:= PneuActIdle;

					tyP0922Stopper.tyInStopperDC.tyBtnUnblk.bRtCompl	:= FALSE;
				END_IF

			ELSIF tyP0922Stopper.tyInStopperDC.tyBtnBlk.bRtCompl = TRUE THEN
				tyP0922Stopper.tyInStopperDC.tyBtnBlk.bValue		:= TRUE;
				tyP0922Stopper.tyInStopperDC.tyBtnUnblk.bValue	:= FALSE;

				eInStopperAct	:= PneuActSetExt;

				IF p_eInStopperStat = PneuActSetExt AND p_eInStopperStatus = Done THEN
					eInStopperAct	:= PneuActIdle;

					tyP0922Stopper.tyInStopperDC.tyBtnBlk.bRtCompl	:= FALSE;
				END_IF
			END_IF

		ELSE
			IF (tyP0922Stopper.tyInStopperDC.tyBtnUnblk.bRtCompl = TRUE) OR (tyP0922Stopper.tyInStopperDC.tyBtnBlk.bRtCompl = TRUE) THEN
				IF (tyP0922Stopper.tyInStopperDC.tyBtnUnblk.bValue = TRUE) AND (tyP0922Stopper.tyInStopperDC.tyBtnBlk.bValue = TRUE) THEN

					eInStopperAct	:= PneuActSetAll;

					IF p_eInStopperStat = PneuActSetAll AND p_eInStopperStatus = Done THEN
						eInStopperAct	:= PneuActIdle;

						tyP0922Stopper.tyInStopperDC.tyBtnUnblk.bRtCompl	:= FALSE;
						tyP0922Stopper.tyInStopperDC.tyBtnBlk.bRtCompl	:= FALSE;
					END_IF

				ELSIF (tyP0922Stopper.tyInStopperDC.tyBtnUnblk.bValue = TRUE) AND (tyP0922Stopper.tyInStopperDC.tyBtnBlk.bValue = FALSE) THEN

					eInStopperAct	:= PneuActSetRet;

					IF p_eInStopperStat = PneuActSetRet AND p_eInStopperStatus = Done THEN

						eInStopperAct	:= PneuActIdle;

						tyP0922Stopper.tyInStopperDC.tyBtnUnblk.bRtCompl	:= FALSE;
						tyP0922Stopper.tyInStopperDC.tyBtnBlk.bRtCompl	:= FALSE;
					END_IF

				ELSIF (tyP0922Stopper.tyInStopperDC.tyBtnUnblk.bValue = FALSE) AND (tyP0922Stopper.tyInStopperDC.tyBtnBlk.bValue = TRUE) THEN

					eInStopperAct	:= PneuActSetExt;

					IF p_eInStopperStat = PneuActSetExt AND p_eInStopperStatus = Done THEN
						eInStopperAct	:= PneuActIdle;

						tyP0922Stopper.tyInStopperDC.tyBtnUnblk.bRtCompl	:= FALSE;
						tyP0922Stopper.tyInStopperDC.tyBtnBlk.bRtCompl	:= FALSE;
					END_IF

				ELSE
					eInStopperAct	:= PneuActRstAll;

					IF p_eInStopperStat = PneuActRstAll AND p_eInStopperStatus = Done THEN
						eInStopperAct	:= PneuActIdle;

						tyP0922Stopper.tyInStopperDC.tyBtnUnblk.bRtCompl	:= FALSE;
						tyP0922Stopper.tyInStopperDC.tyBtnBlk.bRtCompl	:= FALSE;
					END_IF

				END_IF
			END_IF
		END_IF

		//Update Status
		tyP0922Stopper.tyInStopperFB.tyBtnUnblk.bValue		:= FALSE;
		tyP0922Stopper.tyInStopperFB.tyBtnBlk.bValue			:= FALSE;
		tyP0922Stopper.tyInStopperFB.tyBtnUnblk.bRtCompl		:= FALSE;
		tyP0922Stopper.tyInStopperFB.tyBtnBlk.bRtCompl		:= FALSE;

	END_IF

END_ACTION
```

#### Act_OptP0922RstMnl.st
```iecst
ACTION Act_OptP0922RstMnl:

	IF EDGEPOS((bManualMod = FALSE) OR (p_eStopperAStatus = Error)) THEN

		eStopperAAct	:= PneuActIdle;

		tyP0922Stopper.tyStopperADC.tyBtnBlk.bRtCompl	:= FALSE;
		tyP0922Stopper.tyStopperADC.tyBtnBlk.bValue		:= FALSE;
		tyP0922Stopper.tyStopperADC.tyBtnUnblk.bRtCompl	:= FALSE;
		tyP0922Stopper.tyStopperADC.tyBtnUnblk.bValue	:= FALSE;

		tyP0922Stopper.tyStopperAFB.tyBtnBlk.bRtCompl	:= FALSE;
		tyP0922Stopper.tyStopperAFB.tyBtnBlk.bValue		:= FALSE;
		tyP0922Stopper.tyStopperAFB.tyBtnUnblk.bRtCompl	:= FALSE;
		tyP0922Stopper.tyStopperAFB.tyBtnUnblk.bValue	:= FALSE;

	END_IF

	IF EDGEPOS((bManualMod = FALSE) OR (p_eStopperBStatus = Error)) THEN

		eStopperBAct	:= PneuActIdle;

		tyP0922Stopper.tyStopperBDC.tyBtnBlk.bRtCompl	:= FALSE;
		tyP0922Stopper.tyStopperBDC.tyBtnBlk.bValue		:= FALSE;
		tyP0922Stopper.tyStopperBDC.tyBtnUnblk.bRtCompl	:= FALSE;
		tyP0922Stopper.tyStopperBDC.tyBtnUnblk.bValue	:= FALSE;

		tyP0922Stopper.tyStopperBFB.tyBtnBlk.bRtCompl	:= FALSE;
		tyP0922Stopper.tyStopperBFB.tyBtnBlk.bValue		:= FALSE;
		tyP0922Stopper.tyStopperBFB.tyBtnUnblk.bRtCompl	:= FALSE;
		tyP0922Stopper.tyStopperBFB.tyBtnUnblk.bValue	:= FALSE;

	END_IF

	IF EDGEPOS((bManualMod = FALSE) OR (p_eStopperBStatus = Error)) THEN

		eInStopperAct	:= PneuActIdle;

		tyP0922Stopper.tyInStopperDC.tyBtnBlk.bRtCompl	:= FALSE;
		tyP0922Stopper.tyInStopperDC.tyBtnBlk.bValue		:= FALSE;
		tyP0922Stopper.tyInStopperDC.tyBtnUnblk.bRtCompl	:= FALSE;
		tyP0922Stopper.tyInStopperDC.tyBtnUnblk.bValue	:= FALSE;

		tyP0922Stopper.tyInStopperFB.tyBtnBlk.bRtCompl	:= FALSE;
		tyP0922Stopper.tyInStopperFB.tyBtnBlk.bValue		:= FALSE;
		tyP0922Stopper.tyInStopperFB.tyBtnUnblk.bRtCompl	:= FALSE;
		tyP0922Stopper.tyInStopperFB.tyBtnUnblk.bValue	:= FALSE;

	END_IF

	IF EDGEPOS(bManualMod = FALSE) THEN
		tyP0922Stopper.tyStopperACom.tyBtnSwitch.bValue := FALSE;
		tyP0922Stopper.tyStopperBCom.tyBtnSwitch.bValue := FALSE;
		tyP0922Stopper.tyInStopperCom.tyBtnSwitch.bValue := FALSE;

		IF p_tyNtParamCurr.bProjStopperAPrep  THEN
			fUIInRtStatHide(ADR(tyP0922Stopper.tyStopperADC.tyLyr.uiRtStat));
			fUIInRtStatOff(ADR(tyP0922Stopper.tyStopperAFB.tyLyr.uiRtStat));
		END_IF
		IF p_tyNtParamCurr.bProjStopperBPrep THEN
			fUIInRtStatHide(ADR(tyP0922Stopper.tyStopperBDC.tyLyr.uiRtStat));
			fUIInRtStatOff(ADR(tyP0922Stopper.tyStopperBFB.tyLyr.uiRtStat));
		END_IF
		IF p_tyNtParamCurr.bProjInletStopperPrep THEN
			fUIInRtStatHide(ADR(tyP0922Stopper.tyInStopperDC.tyLyr.uiRtStat));
			fUIInRtStatOff(ADR(tyP0922Stopper.tyInStopperFB.tyLyr.uiRtStat));
		END_IF
	END_IF

END_ACTION
```

#### Act_EntP0923Disp.st
```iecst
ACTION Act_EntP0923Disp:

	//Access Address
	IF bDispSafetyBar1 = TRUE THEN

		p_tyC0003DualMask ACCESS ADR(tyP0923SafetyBar.tyDualMaskHide);

		IF p_tyNtParamCurr.eProjMag = ULMagDual THEN
			p_tyC0004Navi ACCESS ADR(tyP0923SafetyBar.tyNaviBack);
		ELSE
			p_tyC0004Navi ACCESS ADR(tyP0923SafetyBar.tyNaviLyr1);
		END_IF

		p_tyC0005Main ACCESS ADR(tyCommon.tyMain);

		p_tyC0007Notif ACCESS ADR(tyCommon.tyNotif);

		p_tyC0008MsgBox ACCESS ADR(tyP0923SafetyBar.tyMsgBoxHide);

		p_tyC0009Info ACCESS ADR(tyCommon.tyInfo);

		p_tyP0923LftSafetyBarCom ACCESS ADR(tyP0923SafetyBar.tyMag1SafetyBarCom);
		p_tyP0923LftSafetyBarDC ACCESS ADR(tyP0923SafetyBar.tyMag1SafetyBarDC);
		p_tyP0923LftSafetyBarFB ACCESS ADR(tyP0923SafetyBar.tyMag1SafetyBarFB);

		p_tyP0923RgtSafetyBarCom ACCESS ADR(tyP0923SafetyBar.tyMag2SafetyBarCom);
		p_tyP0923RgtSafetyBarDC ACCESS ADR(tyP0923SafetyBar.tyMag2SafetyBarDC);
		p_tyP0923RgtSafetyBarFB ACCESS ADR(tyP0923SafetyBar.tyMag2SafetyBarFB);

	ELSIF bDispSafetyBar2 = TRUE THEN

		p_tyC0003DualMask ACCESS ADR(tyP0923SafetyBar.tyDualMaskHide);

		p_tyC0004Navi ACCESS ADR(tyP0923SafetyBar.tyNaviLyr2);

		p_tyC0005Main ACCESS ADR(tyCommon.tyMain);

		p_tyC0007Notif ACCESS ADR(tyCommon.tyNotif);

		p_tyC0008MsgBox ACCESS ADR(tyP0923SafetyBar.tyMsgBoxHide);

		p_tyC0009Info ACCESS ADR(tyCommon.tyInfo);

		p_tyP0923LftSafetyBarCom ACCESS ADR(tyP0923SafetyBar.tyMag3SafetyBarCom);
		p_tyP0923LftSafetyBarDC ACCESS ADR(tyP0923SafetyBar.tyMag3SafetyBarDC);
		p_tyP0923LftSafetyBarFB ACCESS ADR(tyP0923SafetyBar.tyMag3SafetyBarFB);

		p_tyP0923RgtSafetyBarCom ACCESS ADR(tyP0923SafetyBar.tyRgtSafetyBarComHide);
		p_tyP0923RgtSafetyBarDC ACCESS ADR(tyP0923SafetyBar.tyRgtSafetyBarDCHide);
		p_tyP0923RgtSafetyBarFB ACCESS ADR(tyP0923SafetyBar.tyRgtSafetyBarFBHide);

	END_IF

	//Disp
	//Update Status
	tyP0923SafetyBar.tyMag1SafetyBarDC.tyBtnExt.bValue	:= p_bMag1SafetyBarExtCtrl;
	tyP0923SafetyBar.tyMag1SafetyBarDC.tyBtnRet.bValue	:= p_bMag1SafetyBarRetCtrl;
	tyP0923SafetyBar.tyMag2SafetyBarDC.tyBtnExt.bValue	:= p_bMag2SafetyBarExtCtrl;
	tyP0923SafetyBar.tyMag2SafetyBarDC.tyBtnRet.bValue	:= p_bMag2SafetyBarRetCtrl;
	tyP0923SafetyBar.tyMag3SafetyBarDC.tyBtnExt.bValue	:= p_bMag3SafetyBarExtCtrl;
	tyP0923SafetyBar.tyMag3SafetyBarDC.tyBtnRet.bValue	:= p_bMag3SafetyBarRetCtrl;

END_ACTION
```
